C01817=1047.230,-124.087,431.232,169.475,31.897,156.058
C01818=1047.225,-124.336,431.241,169.473,31.897,156.058
C01819=1047.219,-124.586,431.251,169.471,31.897,156.058
C01820=1047.212,-124.836,431.260,169.469,31.897,156.058
C01821=1047.206,-125.086,431.268,169.466,31.896,156.058
C01822=1047.200,-125.335,431.278,169.464,31.897,156.058
C01823=1047.193,-125.585,431.287,169.462,31.897,156.058
C01824=1047.188,-125.835,431.295,169.459,31.897,156.058
C01825=1047.181,-126.085,431.305,169.457,31.897,156.058
C01826=1047.176,-126.335,431.313,169.455,31.897,156.059
C01827=1047.169,-126.584,431.322,169.452,31.897,156.059
C01828=1047.163,-126.834,431.332,169.450,31.896,156.059
C01829=1047.157,-127.084,431.341,169.448,31.897,156.059
C01830=1047.151,-127.333,431.349,169.445,31.896,156.059
C01831=1047.145,-127.583,431.359,169.443,31.897,156.059
C01832=1047.139,-127.833,431.367,169.441,31.897,156.059
C01833=1047.133,-128.082,431.377,169.439,31.896,156.059
C01834=1047.129,-128.332,431.387,169.436,31.895,156.059
C01835=1047.126,-128.582,431.398,169.434,31.894,156.059
C01836=1047.124,-128.832,431.410,169.432,31.892,156.059
C01837=1047.122,-129.082,431.421,169.432,31.890,156.058
C01838=1047.123,-129.332,431.434,169.430,31.887,156.058
C01839=1047.123,-129.583,431.447,169.428,31.883,156.058
C01840=1047.124,-129.832,431.461,169.427,31.880,156.057
C01841=1047.127,-130.083,431.476,169.426,31.876,156.056
C01842=1047.131,-130.334,431.492,169.424,31.871,156.056
C01843=1047.135,-130.585,431.507,169.423,31.866,156.055
C01844=1047.141,-130.835,431.523,169.423,31.861,156.054
C01845=1047.146,-131.085,431.541,169.422,31.854,156.053
C01846=1046.788,-131.108,431.305,169.376,32.030,156.085
C01847=1046.781,-130.858,431.288,169.377,32.036,156.086
C01848=1046.776,-130.609,431.271,169.378,32.042,156.087
C01849=1046.771,-130.358,431.256,169.379,32.047,156.088
C01850=1046.769,-130.107,431.240,169.380,32.051,156.089
C01851=1046.765,-129.857,431.226,169.381,32.055,156.089
C01852=1046.764,-129.607,431.212,169.383,32.059,156.090
C01853=1046.763,-129.356,431.198,169.383,32.063,156.090
C01854=1046.763,-129.106,431.186,169.385,32.065,156.091
C01855=1046.765,-128.856,431.173,169.387,32.068,156.091
C01856=1046.767,-128.606,431.162,169.389,32.070,156.091
C01857=1046.771,-128.356,431.151,169.391,32.071,156.092
C01858=1046.775,-128.106,431.141,169.393,32.072,156.092
C01859=1046.779,-127.856,431.131,169.395,32.072,156.092
C01860=1046.786,-127.607,431.122,169.397,32.073,156.091
C01861=1046.791,-127.357,431.113,169.400,32.072,156.091
C01862=1046.798,-127.107,431.104,169.402,32.072,156.091
C01863=1046.803,-126.858,431.095,169.404,32.072,156.091
C01864=1046.809,-126.608,431.086,169.407,32.072,156.091
C01865=1046.816,-126.358,431.077,169.409,32.072,156.091
C01866=1046.822,-126.108,431.069,169.411,32.072,156.091
C01867=1046.828,-125.859,431.059,169.414,32.072,156.091
C01868=1046.834,-125.609,431.050,169.416,32.072,156.091
C01869=1046.840,-125.359,431.042,169.418,32.072,156.090
C01870=1046.847,-125.109,431.032,169.420,32.072,156.090
C01871=1046.853,-124.860,431.024,169.422,32.072,156.090
C01872=1046.859,-124.610,431.014,169.424,32.072,156.090
C01873=1046.865,-124.360,431.005,169.427,32.072,156.090
C01874=1046.871,-124.110,430.996,169.429,32.072,156.090
C01875=1046.877,-123.861,430.987,169.431,32.072,156.090
C01876=1046.883,-123.611,430.978,169.434,32.073,156.090
C01877=1046.889,-123.361,430.968,169.436,32.072,156.090
C01878=1046.895,-123.111,430.959,169.438,32.072,156.090
C01879=1046.901,-122.862,430.950,169.441,32.073,156.089
C01880=1046.907,-122.612,430.941,169.443,32.072,156.089
C01881=1046.914,-122.362,430.932,169.445,32.073,156.089
C01882=1046.920,-122.112,430.923,169.448,32.073,156.089
C01883=1046.926,-121.862,430.913,169.450,32.073,156.089
C01884=1046.932,-121.613,430.904,169.452,32.073,156.089
C01885=1046.937,-121.363,430.895,169.455,32.073,156.089
C01886=1046.944,-121.113,430.886,169.457,32.073,156.089
C01887=1046.950,-120.864,430.877,169.459,32.073,156.089
C01888=1046.957,-120.614,430.867,169.462,32.073,156.089
C01889=1046.962,-120.365,430.858,169.464,32.074,156.088
C01890=1046.968,-120.114,430.849,169.466,32.074,156.088
C01891=1046.974,-119.864,430.840,169.469,32.074,156.088
C01892=1046.980,-119.615,430.830,169.471,32.074,156.088
C01893=1046.987,-119.365,430.820,169.472,32.074,156.088
C01894=1046.993,-119.115,430.811,169.475,32.075,156.088
C01895=1046.999,-118.866,430.802,169.477,32.075,156.088
C01896=1047.005,-118.616,430.793,169.479,32.074,156.088
C01897=1047.011,-118.366,430.784,169.482,32.075,156.088
C01898=1047.017,-118.116,430.774,169.484,32.075,156.088
C01899=1047.023,-117.866,430.765,169.486,32.075,156.088
C01900=1047.030,-117.617,430.755,169.489,32.076,156.088
C01901=1047.036,-117.367,430.746,169.491,32.075,156.087
C01902=1047.041,-117.118,430.736,169.493,32.075,156.087
C01903=1047.048,-116.868,430.727,169.496,32.076,156.087
C01904=1047.054,-116.618,430.717,169.498,32.076,156.087
C01905=1047.060,-116.368,430.708,169.500,32.076,156.087
C01906=1047.066,-116.119,430.698,169.502,32.076,156.087
C01907=1047.073,-115.833,430.688,169.505,32.077,156.087
C01908=1047.080,-115.547,430.677,169.508,32.077,156.087
C01909=1047.087,-115.262,430.666,169.510,32.077,156.087
C01910=1047.095,-114.976,430.656,169.513,32.077,156.087
C01911=1047.101,-114.726,430.646,169.515,32.077,156.087
C01912=1047.107,-114.476,430.637,169.518,32.078,156.087
C01913=1047.113,-114.226,430.627,169.519,32.078,156.087
C01914=1047.119,-113.977,430.617,169.521,32.078,156.087
C01915=1047.125,-113.727,430.608,169.524,32.079,156.086
C01916=1047.130,-113.477,430.598,169.526,32.079,156.086
C01917=1047.137,-113.228,430.588,169.528,32.079,156.086
C01918=1047.143,-112.978,430.578,169.531,32.079,156.086
C01919=1047.149,-112.729,430.569,169.533,32.080,156.086
C01920=1047.155,-112.479,430.559,169.535,32.080,156.086
C01921=1047.161,-112.229,430.550,169.537,32.080,156.086
C01922=1047.168,-111.979,430.540,169.540,32.080,156.086
C01923=1047.174,-111.729,430.530,169.542,32.081,156.086
C01924=1047.180,-111.480,430.521,169.544,32.081,156.086
C01925=1047.186,-111.230,430.511,169.547,32.081,156.086
C01926=1047.192,-110.980,430.502,169.549,32.082,156.086
C01927=1047.198,-110.730,430.492,169.551,32.082,156.086
C01928=1047.205,-110.481,430.482,169.554,32.082,156.086
C01929=1047.210,-110.231,430.472,169.556,32.082,156.086
C01930=1047.216,-109.981,430.462,169.558,32.083,156.086
C01931=1047.223,-109.731,430.453,169.560,32.083,156.085
C01932=1047.229,-109.481,430.443,169.563,32.083,156.085
C01933=1047.235,-109.232,430.433,169.565,32.083,156.085
C01934=1047.241,-108.983,430.423,169.566,32.084,156.085
C01935=1047.248,-108.733,430.414,169.569,32.084,156.085
C01936=1047.254,-108.483,430.404,169.571,32.085,156.085
C01937=1047.260,-108.233,430.394,169.573,32.085,156.085
C01938=1047.265,-107.983,430.384,169.576,32.086,156.085
C01939=1047.272,-107.734,430.374,169.578,32.086,156.085
C01940=1047.278,-107.484,430.364,169.580,32.086,156.085
C01941=1047.284,-107.234,430.355,169.582,32.086,156.085
C01942=1047.290,-106.984,430.345,169.585,32.087,156.085
C01943=1047.297,-106.735,430.335,169.587,32.087,156.085
C01944=1047.302,-106.485,430.325,169.589,32.088,156.085
C01945=1047.309,-106.235,430.315,169.592,32.088,156.085
C01946=1047.315,-105.986,430.305,169.594,32.088,156.085
C01947=1047.321,-105.736,430.295,169.596,32.089,156.085
C01948=1047.327,-105.486,430.285,169.598,32.089,156.085
C01949=1047.334,-105.236,430.275,169.601,32.090,156.085
C01950=1047.340,-104.987,430.265,169.603,32.090,156.085
C01951=1047.346,-104.737,430.255,169.605,32.090,156.085
C01952=1047.352,-104.487,430.245,169.608,32.091,156.085
C01953=1047.358,-104.238,430.235,169.609,32.092,156.085
C01954=1047.364,-103.988,430.225,169.611,32.092,156.085
C01955=1047.370,-103.738,430.215,169.613,32.092,156.085
C01956=1047.376,-103.488,430.205,169.616,32.092,156.084
C01957=1047.382,-103.239,430.195,169.618,32.093,156.084
C01958=1047.388,-102.989,430.185,169.620,32.093,156.084
C01959=1047.394,-102.739,430.175,169.622,32.094,156.084
C01960=1047.401,-102.489,430.164,169.625,32.095,156.084
C01961=1047.407,-102.240,430.155,169.627,32.095,156.084
C01962=1047.413,-101.990,430.144,169.629,32.095,156.084
C01963=1047.419,-101.740,430.134,169.632,32.096,156.084
C01964=1047.425,-101.491,430.125,169.634,32.096,156.084
C01965=1047.431,-101.241,430.114,169.636,32.097,156.084
C01966=1047.437,-100.991,430.104,169.638,32.097,156.084
C01967=1047.444,-100.742,430.094,169.641,32.098,156.084
C01968=1047.450,-100.491,430.084,169.643,32.098,156.084
C01969=1047.456,-100.242,430.073,169.645,32.098,156.084
C01970=1047.462,-99.992,430.064,169.647,32.099,156.084
C01971=1047.469,-99.705,430.051,169.650,32.100,156.084
C01972=1047.476,-99.419,430.040,169.652,32.101,156.084
C01973=1047.484,-99.132,430.028,169.654,32.101,156.084
C01974=1047.491,-98.846,430.017,169.657,32.101,156.084
C01975=1047.496,-98.597,430.006,169.659,32.102,156.084
C01976=1047.503,-98.346,429.996,169.661,32.102,156.084
C01977=1047.510,-98.097,429.986,169.664,32.103,156.084
C01978=1047.515,-97.847,429.975,169.666,32.103,156.084
C01979=1047.522,-97.598,429.965,169.668,32.104,156.084
C01980=1047.528,-97.347,429.955,169.670,32.105,156.084
C01981=1047.534,-97.098,429.944,169.673,32.105,156.084
C01982=1047.540,-96.848,429.933,169.675,32.106,156.084
C01983=1047.546,-96.598,429.924,169.677,32.106,156.084
C01984=1047.552,-96.349,429.913,169.679,32.107,156.084
C01985=1047.558,-96.099,429.902,169.682,32.108,156.084
C01986=1047.564,-95.849,429.892,169.684,32.108,156.084
C01987=1047.570,-95.599,429.881,169.686,32.109,156.084
C01988=1047.577,-95.350,429.871,169.688,32.109,156.084
C01989=1047.582,-95.100,429.861,169.691,32.110,156.084
C01990=1047.588,-94.851,429.851,169.692,32.110,156.084
C01991=1047.595,-94.601,429.839,169.694,32.111,156.084
C01992=1047.600,-94.351,429.829,169.696,32.112,156.084
C01993=1047.607,-94.101,429.819,169.699,32.113,156.084
C01994=1047.612,-93.852,429.808,169.701,32.113,156.084
C01995=1047.619,-93.602,429.797,169.703,32.114,156.084
C01996=1047.625,-93.352,429.787,169.705,32.115,156.084
C01997=1047.631,-93.102,429.776,169.707,32.115,156.084
C01998=1047.637,-92.853,429.766,169.710,32.116,156.084
C01999=1047.643,-92.603,429.755,169.712,32.117,156.084
C02000=1047.649,-92.353,429.745,169.714,32.117,156.084
C02001=1047.655,-92.104,429.734,169.716,32.118,156.084
C02002=1047.661,-91.854,429.724,169.719,32.119,156.084
C02003=1047.668,-91.604,429.713,169.721,32.119,156.084
C02004=1047.674,-91.355,429.702,169.723,32.120,156.084
C02005=1047.679,-91.105,429.692,169.725,32.121,156.084
C02006=1047.686,-90.855,429.681,169.728,32.121,156.084
C02007=1047.692,-90.605,429.670,169.730,32.122,156.084
C02008=1047.698,-90.356,429.659,169.731,32.123,156.084
C02009=1047.704,-90.107,429.649,169.733,32.123,156.084
C02010=1047.711,-89.857,429.638,169.735,32.124,156.084
C02011=1047.716,-89.607,429.627,169.738,32.125,156.084
C02012=1047.723,-89.357,429.617,169.740,32.125,156.084
C02013=1047.729,-89.107,429.606,169.742,32.126,156.084
C02014=1047.735,-88.858,429.596,169.744,32.127,156.084
C02015=1047.741,-88.608,429.585,169.747,32.127,156.084
C02016=1047.748,-88.358,429.574,169.749,32.128,156.084
C02017=1047.754,-88.109,429.564,169.751,32.129,156.084
C02018=1047.760,-87.859,429.552,169.753,32.129,156.084
C02019=1047.766,-87.609,429.541,169.756,32.130,156.084
C02020=1047.773,-87.360,429.531,169.758,32.131,156.084
C02021=1047.779,-87.110,429.520,169.760,32.132,156.085
C02022=1047.785,-86.860,429.509,169.762,32.132,156.084
C02023=1047.791,-86.611,429.499,169.764,32.133,156.085
C02024=1047.797,-86.361,429.487,169.767,32.134,156.085
C02025=1047.803,-86.111,429.477,169.768,32.135,156.085
C02026=1047.810,-85.861,429.467,169.770,32.135,156.085
C02027=1047.816,-85.612,429.456,169.772,32.136,156.085
C02028=1047.821,-85.362,429.445,169.774,32.137,156.085
C02029=1047.828,-85.112,429.434,169.777,32.137,156.085
C02030=1047.835,-84.863,429.423,169.779,32.138,156.085
C02031=1047.841,-84.613,429.411,169.781,32.139,156.085
C02032=1047.847,-84.364,429.401,169.783,32.140,156.085
C02033=1047.854,-84.114,429.390,169.786,32.141,156.085
C02034=1047.860,-83.864,429.379,169.788,32.141,156.085
C02035=1047.866,-83.580,429.367,169.790,32.142,156.085
C02036=1047.874,-83.295,429.354,169.793,32.143,156.085
C02037=1047.881,-83.011,429.341,169.795,32.144,156.085
C02038=1047.888,-82.726,429.329,169.798,32.145,156.085
C02039=1047.895,-82.476,429.319,169.800,32.146,156.085
C02040=1047.900,-82.227,429.308,169.802,32.146,156.085
C02041=1047.907,-81.977,429.296,169.804,32.147,156.085
C02042=1047.913,-81.728,429.285,169.807,32.148,156.085
C02043=1047.920,-81.478,429.274,169.808,32.148,156.085
C02044=1047.926,-81.229,429.264,169.810,32.149,156.085
C02045=1047.932,-80.978,429.252,169.812,32.150,156.085
C02046=1047.938,-80.729,429.242,169.815,32.151,156.085
C02047=1047.945,-80.479,429.231,169.817,32.151,156.085
C02048=1047.951,-80.230,429.219,169.819,32.152,156.085
C02049=1047.957,-79.980,429.208,169.821,32.153,156.085
C02050=1047.964,-79.731,429.198,169.823,32.154,156.085
C02051=1047.970,-79.481,429.186,169.826,32.155,156.085
C02052=1047.976,-79.231,429.176,169.828,32.156,156.086
C02053=1047.982,-78.981,429.164,169.830,32.157,156.086
C02054=1047.988,-78.732,429.153,169.832,32.158,156.086
C02055=1047.994,-78.482,429.142,169.834,32.158,156.086
C02056=1048.000,-78.232,429.131,169.836,32.159,156.086
C02057=1048.007,-77.983,429.119,169.839,32.160,156.086
C02058=1048.013,-77.733,429.108,169.841,32.161,156.086
C02059=1048.019,-77.483,429.097,169.843,32.162,156.086
C02060=1048.025,-77.234,429.085,169.844,32.163,156.086
C02061=1048.031,-76.984,429.074,169.846,32.164,156.086
C02062=1048.037,-76.734,429.063,169.848,32.165,156.086
C02063=1048.044,-76.485,429.051,169.851,32.166,156.086
C02064=1048.049,-76.235,429.040,169.853,32.166,156.086
C02065=1048.056,-75.985,429.029,169.855,32.167,156.086
C02066=1048.062,-75.736,429.017,169.857,32.168,156.086
C02067=1048.068,-75.486,429.006,169.859,32.169,156.086
C02068=1048.075,-75.236,428.995,169.862,32.170,156.086
C02069=1048.081,-74.987,428.983,169.864,32.171,156.086
C02070=1048.087,-74.737,428.972,169.866,32.172,156.087
C02071=1048.093,-74.487,428.961,169.868,32.173,156.087
C02072=1048.099,-74.238,428.949,169.870,32.173,156.087
C02073=1048.106,-73.988,428.938,169.872,32.174,156.087
C02074=1048.112,-73.739,428.926,169.875,32.175,156.087
C02075=1048.118,-73.489,428.915,169.877,32.177,156.087
C02076=1048.124,-73.240,428.903,169.879,32.178,156.087
C02077=1048.130,-72.989,428.892,169.880,32.178,156.087
C02078=1048.135,-72.740,428.881,169.882,32.179,156.087
C02079=1048.142,-72.490,428.869,169.884,32.181,156.087
C02080=1048.148,-72.241,428.858,169.886,32.182,156.087
C02081=1048.154,-71.991,428.845,169.889,32.183,156.087
C02082=1048.160,-71.741,428.834,169.891,32.184,156.087
C02083=1048.166,-71.492,428.822,169.893,32.185,156.088
C02084=1048.172,-71.242,428.811,169.895,32.186,156.088
C02085=1048.178,-70.993,428.800,169.897,32.187,156.088
C02086=1048.184,-70.743,428.787,169.899,32.188,156.088
C02087=1048.191,-70.493,428.776,169.901,32.189,156.088
C02088=1048.197,-70.244,428.764,169.903,32.190,156.088
C02089=1048.203,-69.994,428.753,169.906,32.191,156.088
C02090=1048.208,-69.744,428.741,169.908,32.192,156.088
C02091=1048.215,-69.494,428.729,169.910,32.193,156.088
C02092=1048.221,-69.245,428.718,169.912,32.194,156.088
C02093=1048.227,-68.995,428.705,169.913,32.195,156.088
C02094=1048.233,-68.745,428.694,169.915,32.196,156.089
C02095=1048.240,-68.496,428.682,169.917,32.197,156.089
C02096=1048.245,-68.246,428.671,169.920,32.198,156.089
C02097=1048.251,-67.996,428.659,169.922,32.200,156.089
C02098=1048.258,-67.747,428.647,169.924,32.201,156.089
C02099=1048.264,-67.465,428.634,169.926,32.201,156.089
C02100=1048.271,-67.183,428.620,169.929,32.203,156.089
C02101=1048.278,-66.900,428.607,169.931,32.204,156.089
C02102=1048.286,-66.618,428.594,169.933,32.205,156.089
C02103=1048.292,-66.368,428.582,169.936,32.206,156.089
C02104=1048.298,-66.118,428.571,169.938,32.208,156.090
C02105=1048.304,-65.869,428.559,169.940,32.209,156.090
C02106=1048.310,-65.619,428.546,169.942,32.210,156.090
C02107=1048.316,-65.369,428.535,169.944,32.211,156.090
C02108=1048.322,-65.120,428.524,169.946,32.212,156.090
C02109=1048.329,-64.871,428.512,169.948,32.213,156.090
C02110=1048.335,-64.621,428.499,169.949,32.214,156.090
C02111=1048.341,-64.371,428.488,169.951,32.215,156.090
C02112=1048.347,-64.122,428.476,169.954,32.216,156.090
C02113=1048.353,-63.872,428.464,169.956,32.218,156.090
C02114=1048.360,-63.622,428.452,169.958,32.218,156.090
C02115=1048.366,-63.372,428.440,169.960,32.219,156.091
C02116=1048.371,-63.123,428.428,169.962,32.221,156.091
C02117=1048.378,-62.873,428.416,169.964,32.222,156.091
C02118=1048.385,-62.624,428.404,169.966,32.223,156.091
C02119=1048.391,-62.374,428.392,169.968,32.224,156.091
C02120=1048.397,-62.124,428.381,169.971,32.225,156.091
C02121=1048.403,-61.875,428.369,169.973,32.226,156.091
C02122=1048.409,-61.625,428.356,169.975,32.227,156.091
C02123=1048.416,-61.376,428.344,169.977,32.229,156.091
C02124=1048.422,-61.126,428.332,169.979,32.230,156.092
C02125=1048.428,-60.876,428.320,169.981,32.231,156.092
C02126=1048.434,-60.627,428.308,169.982,32.232,156.092
C02127=1048.441,-60.377,428.297,169.984,32.233,156.092
C02128=1048.446,-60.127,428.284,169.986,32.234,156.092
C02129=1048.453,-59.878,428.273,169.988,32.235,156.092
C02130=1048.460,-59.628,428.261,169.991,32.236,156.092
C02131=1048.465,-59.379,428.248,169.993,32.238,156.092
C02132=1048.472,-59.129,428.236,169.995,32.238,156.092
C02133=1048.478,-58.880,428.224,169.997,32.240,156.093
C02134=1048.484,-58.630,428.212,169.999,32.241,156.093
C02135=1048.491,-58.380,428.200,170.001,32.242,156.093
C02136=1048.497,-58.130,428.187,170.003,32.243,156.093
C02137=1048.503,-57.881,428.175,170.005,32.244,156.093
C02138=1048.510,-57.631,428.163,170.007,32.246,156.093
C02139=1048.515,-57.382,428.151,170.009,32.246,156.093
C02140=1048.522,-57.132,428.139,170.012,32.248,156.093
C02141=1048.529,-56.883,428.127,170.014,32.249,156.093
C02142=1048.535,-56.633,428.115,170.016,32.250,156.094
C02143=1048.545,-56.216,428.094,170.018,32.252,156.094
C02144=1048.555,-55.799,428.074,170.022,32.254,156.094
C02145=1048.566,-55.381,428.054,170.025,32.256,156.094
C02146=1048.577,-54.964,428.034,170.029,32.258,156.094
C02147=1048.584,-54.714,428.022,170.031,32.259,156.094
C02148=1048.589,-54.465,428.009,170.033,32.260,156.095
C02149=1048.596,-54.215,427.997,170.035,32.261,156.095
C02150=1048.603,-53.965,427.985,170.037,32.262,156.095
C02151=1048.608,-53.716,427.973,170.039,32.264,156.095
C02152=1048.615,-53.467,427.961,170.041,32.265,156.095
C02153=1048.621,-53.217,427.948,170.043,32.266,156.095
C02154=1048.628,-52.968,427.936,170.045,32.267,156.095
C02155=1048.634,-52.718,427.924,170.047,32.268,156.095
C02156=1048.640,-52.468,427.911,170.050,32.269,156.095
C02157=1048.647,-52.219,427.899,170.051,32.271,156.096
C02158=1048.653,-51.969,427.887,170.053,32.272,156.096
C02159=1048.663,-51.606,427.869,170.056,32.274,156.096
C02160=1048.671,-51.243,427.851,170.059,32.275,156.096
C02161=1048.681,-50.880,427.833,170.062,32.277,156.096
C02162=1048.691,-50.517,427.815,170.065,32.279,156.096
C02163=1048.697,-50.267,427.802,170.067,32.280,156.096
C02164=1048.703,-50.017,427.790,170.069,32.282,156.097
C02165=1048.709,-49.767,427.777,170.071,32.283,156.097
C02166=1048.716,-49.518,427.764,170.073,32.284,156.097
C02167=1048.722,-49.268,427.752,170.075,32.285,156.097
C02168=1048.728,-49.018,427.739,170.077,32.287,156.097
C02169=1048.733,-48.768,427.727,170.079,32.288,156.097
C02170=1048.740,-48.520,427.714,170.081,32.289,156.097
C02171=1048.746,-48.270,427.702,170.083,32.291,156.098
C02172=1048.752,-48.020,427.689,170.084,32.292,156.098
C02173=1048.758,-47.771,427.676,170.086,32.294,156.098
C02174=1048.764,-47.522,427.664,170.088,32.294,156.098
C02175=1048.770,-47.272,427.652,170.090,32.296,156.098
C02176=1048.777,-47.022,427.638,170.092,32.297,156.098
C02177=1048.782,-46.773,427.626,170.094,32.299,156.099
C02178=1048.790,-46.522,427.613,170.096,32.300,156.099
C02179=1048.796,-46.273,427.600,170.098,32.301,156.099
C02180=1048.802,-46.023,427.588,170.100,32.303,156.099
C02181=1048.808,-45.774,427.574,170.102,32.304,156.099
C02182=1048.814,-45.524,427.562,170.104,32.306,156.099
C02183=1048.821,-45.274,427.550,170.107,32.307,156.099
C02184=1048.827,-45.025,427.537,170.109,32.308,156.100
C02185=1048.833,-44.775,427.524,170.111,32.310,156.100
C02186=1048.839,-44.526,427.511,170.113,32.311,156.100
C02187=1048.846,-44.276,427.499,170.115,32.312,156.100
C02188=1048.852,-44.027,427.485,170.117,32.313,156.100
C02189=1048.858,-43.777,427.473,170.118,32.315,156.100
C02190=1048.864,-43.527,427.460,170.120,32.316,156.101
C02191=1048.870,-43.278,427.447,170.122,32.318,156.101
C02192=1048.877,-43.029,427.435,170.124,32.319,156.101
C02193=1048.883,-42.779,427.422,170.126,32.320,156.101
C02194=1048.889,-42.529,427.409,170.128,32.322,156.101
C02195=1048.895,-42.279,427.396,170.130,32.323,156.101
C02196=1048.901,-42.030,427.383,170.132,32.324,156.101
C02197=1048.908,-41.781,427.370,170.134,32.326,156.102
C02198=1048.914,-41.531,427.358,170.136,32.327,156.102
C02199=1048.920,-41.281,427.345,170.138,32.328,156.102
C02200=1048.927,-41.032,427.331,170.140,32.330,156.102
C02201=1048.933,-40.782,427.319,170.142,32.331,156.102
C02202=1048.939,-40.532,427.305,170.144,32.333,156.102
C02203=1048.946,-40.283,427.293,170.146,32.334,156.103
C02204=1048.952,-40.034,427.280,170.148,32.335,156.103
C02205=1048.958,-39.784,427.267,170.150,32.336,156.103
C02206=1048.964,-39.534,427.254,170.152,32.338,156.103
C02207=1048.971,-39.285,427.241,170.153,32.339,156.103
C02208=1048.977,-39.035,427.228,170.155,32.341,156.103
C02209=1048.984,-38.786,427.215,170.157,32.342,156.104
C02210=1048.990,-38.536,427.203,170.159,32.344,156.104
C02211=1048.996,-38.286,427.189,170.161,32.345,156.104
C02212=1049.002,-38.037,427.176,170.163,32.347,156.104
C02213=1049.008,-37.787,427.163,170.165,32.348,156.104
C02214=1049.014,-37.537,427.149,170.167,32.350,156.104
C02215=1049.021,-37.288,427.136,170.169,32.351,156.105
C02216=1049.026,-37.038,427.124,170.171,32.353,156.105
C02217=1049.033,-36.789,427.110,170.173,32.354,156.105
C02218=1049.039,-36.539,427.097,170.175,32.356,156.105
C02219=1049.045,-36.290,427.084,170.177,32.357,156.105
C02220=1049.051,-36.040,427.071,170.179,32.359,156.105
C02221=1049.058,-35.790,427.058,170.181,32.360,156.106
C02222=1049.064,-35.541,427.044,170.183,32.361,156.106
C02223=1049.071,-35.261,427.030,170.185,32.363,156.106
C02224=1049.078,-34.980,427.015,170.186,32.364,156.106
C02225=1049.085,-34.699,427.000,170.188,32.366,156.106
C02226=1049.092,-34.419,426.985,170.190,32.368,156.107
C02227=1049.098,-34.170,426.972,170.192,32.369,156.107
C02228=1049.104,-33.920,426.958,170.194,32.371,156.107
C02229=1049.110,-33.671,426.946,170.196,32.372,156.107
C02230=1049.117,-33.421,426.932,170.198,32.374,156.107
C02231=1049.123,-33.171,426.919,170.200,32.375,156.108
C02232=1049.129,-32.922,426.906,170.202,32.377,156.108
C02233=1049.135,-32.673,426.892,170.204,32.378,156.108
C02234=1049.142,-32.423,426.878,170.206,32.380,156.108
C02235=1049.148,-32.173,426.866,170.208,32.381,156.108
C02236=1049.154,-31.923,426.852,170.210,32.383,156.108
C02237=1049.161,-31.673,426.839,170.212,32.384,156.109
C02238=1049.167,-31.424,426.825,170.214,32.386,156.109
C02239=1049.173,-31.175,426.812,170.216,32.387,156.109
C02240=1049.179,-30.926,426.799,170.218,32.388,156.109
C02241=1049.186,-30.676,426.785,170.219,32.390,156.109
C02242=1049.192,-30.426,426.772,170.221,32.391,156.109
C02243=1049.198,-30.177,426.758,170.223,32.393,156.110
C02244=1049.204,-29.926,426.745,170.225,32.394,156.110
C02245=1049.211,-29.677,426.732,170.227,32.396,156.110
C02246=1049.217,-29.428,426.719,170.229,32.398,156.110
C02247=1049.223,-29.178,426.705,170.231,32.399,156.110
C02248=1049.230,-28.928,426.692,170.233,32.401,156.111
C02249=1049.236,-28.679,426.678,170.235,32.402,156.111
C02250=1049.242,-28.430,426.665,170.236,32.404,156.111
C02251=1049.248,-28.180,426.651,170.238,32.405,156.111
C02252=1049.255,-27.930,426.638,170.240,32.407,156.111
C02253=1049.261,-27.680,426.624,170.242,32.408,156.112
C02254=1049.268,-27.431,426.611,170.244,32.409,156.112
C02255=1049.274,-27.182,426.598,170.246,32.411,156.112
C02256=1049.281,-26.932,426.584,170.248,32.412,156.112
C02257=1049.286,-26.682,426.570,170.250,32.414,156.112
C02258=1049.292,-26.433,426.557,170.252,32.416,156.113
C02259=1049.299,-26.183,426.543,170.253,32.417,156.113
C02260=1049.305,-25.934,426.529,170.255,32.419,156.113
C02261=1049.311,-25.684,426.516,170.257,32.420,156.113
C02262=1049.318,-25.435,426.502,170.259,32.422,156.113
C02263=1049.323,-25.185,426.488,170.261,32.424,156.114
C02264=1049.330,-24.936,426.475,170.263,32.425,156.114
C02265=1049.336,-24.686,426.460,170.264,32.427,156.114
C02266=1049.342,-24.437,426.447,170.266,32.428,156.114
C02267=1049.348,-24.187,426.434,170.268,32.430,156.114
C02268=1049.354,-23.937,426.420,170.270,32.432,156.115
C02269=1049.360,-23.688,426.406,170.272,32.433,156.115
C02270=1049.367,-23.439,426.392,170.274,32.435,156.115
C02271=1049.373,-23.189,426.378,170.276,32.437,156.115
C02272=1049.379,-22.940,426.365,170.278,32.438,156.115
C02273=1049.385,-22.689,426.351,170.280,32.440,156.116
C02274=1049.391,-22.440,426.337,170.282,32.441,156.116
C02275=1049.398,-22.191,426.323,170.284,32.443,156.116
C02276=1049.404,-21.941,426.309,170.285,32.444,156.116
C02277=1049.410,-21.692,426.296,170.287,32.446,156.116
C02278=1049.416,-21.442,426.282,170.288,32.447,156.117
C02279=1049.423,-21.192,426.268,170.290,32.449,156.117
C02280=1049.430,-20.943,426.254,170.292,32.451,156.117
C02281=1049.435,-20.693,426.240,170.294,32.452,156.117
C02282=1049.441,-20.444,426.227,170.296,32.454,156.117
C02283=1049.447,-20.194,426.213,170.298,32.456,156.118
C02284=1049.454,-19.945,426.199,170.300,32.457,156.118
C02285=1049.461,-19.695,426.185,170.302,32.459,156.118
C02286=1049.466,-19.446,426.171,170.303,32.460,156.118
C02287=1049.473,-19.165,426.155,170.306,32.462,156.119
C02288=1049.480,-18.883,426.140,170.308,32.464,156.119
C02289=1049.488,-18.602,426.124,170.310,32.466,156.119
C02290=1049.495,-18.321,426.108,170.312,32.468,156.119
C02291=1049.501,-18.071,426.094,170.314,32.469,156.120
C02292=1049.508,-17.822,426.080,170.316,32.471,156.120
C02293=1049.513,-17.572,426.066,170.318,32.472,156.120
C02294=1049.520,-17.322,426.053,170.320,32.474,156.120
C02295=1049.527,-17.074,426.039,170.321,32.476,156.120
C02296=1049.533,-16.823,426.024,170.323,32.477,156.121
C02297=1049.539,-16.574,426.011,170.324,32.479,156.121
C02298=1049.545,-16.325,425.996,170.326,32.481,156.121
C02299=1049.552,-16.075,425.983,170.328,32.482,156.121
C02300=1049.558,-15.826,425.968,170.330,32.484,156.121
C02301=1049.564,-15.576,425.955,170.332,32.486,156.122
C02302=1049.570,-15.326,425.940,170.334,32.487,156.122
C02303=1049.577,-15.077,425.926,170.336,32.489,156.122
C02304=1049.583,-14.827,425.912,170.337,32.491,156.122
C02305=1049.590,-14.578,425.898,170.339,32.492,156.123
C02306=1049.595,-14.328,425.884,170.341,32.494,156.123
C02307=1049.602,-14.079,425.869,170.343,32.496,156.123
C02308=1049.608,-13.829,425.856,170.345,32.497,156.123
C02309=1049.614,-13.580,425.841,170.347,32.499,156.123
C02310=1049.620,-13.330,425.827,170.349,32.501,156.124
C02311=1049.627,-13.081,425.813,170.350,32.503,156.124
C02312=1049.633,-12.831,425.799,170.352,32.504,156.124
C02313=1049.639,-12.582,425.784,170.354,32.506,156.124
C02314=1049.645,-12.332,425.771,170.356,32.508,156.125
C02315=1049.652,-12.083,425.756,170.358,32.509,156.125
C02316=1049.657,-11.833,425.742,170.359,32.511,156.125
C02317=1049.663,-11.583,425.727,170.361,32.513,156.125
C02318=1049.670,-11.334,425.714,170.362,32.515,156.126
C02319=1049.676,-11.084,425.699,170.364,32.516,156.126
C02320=1049.682,-10.835,425.684,170.366,32.518,156.126
C02321=1049.689,-10.586,425.670,170.368,32.520,156.126
C02322=1049.695,-10.336,425.655,170.370,32.521,156.126
C02323=1049.700,-10.086,425.642,170.372,32.523,156.127
C02324=1049.708,-9.837,425.627,170.374,32.524,156.127
C02325=1049.714,-9.587,425.612,170.375,32.526,156.127
C02326=1049.719,-9.338,425.598,170.377,32.528,156.127
C02327=1049.727,-9.088,425.584,170.379,32.530,156.128
C02328=1049.732,-8.839,425.570,170.381,32.531,156.128
C02329=1049.738,-8.589,425.555,170.383,32.533,156.128
C02330=1049.745,-8.339,425.540,170.385,32.535,156.128
C02331=1049.751,-8.091,425.526,170.386,32.536,156.129
C02332=1049.757,-7.841,425.512,170.388,32.538,156.129
C02333=1049.763,-7.592,425.498,170.390,32.540,156.129
C02334=1049.770,-7.342,425.483,170.392,32.542,156.129
C02335=1049.776,-7.092,425.469,170.394,32.543,156.130
C02336=1049.782,-6.843,425.454,170.396,32.545,156.130
C02337=1049.789,-6.593,425.439,170.396,32.547,156.130
C02338=1049.796,-6.344,425.425,170.398,32.549,156.130
C02339=1049.801,-6.094,425.411,170.400,32.550,156.131
C02340=1049.808,-5.845,425.396,170.402,32.552,156.131
C02341=1049.814,-5.595,425.381,170.404,32.554,156.131
C02342=1049.820,-5.346,425.368,170.406,32.555,156.131
C02343=1049.826,-5.096,425.353,170.407,32.557,156.131
C02344=1049.833,-4.847,425.338,170.409,32.559,156.132
C02345=1049.839,-4.598,425.324,170.411,32.561,156.132
C02346=1049.846,-4.348,425.309,170.413,32.562,156.132
C02347=1049.852,-4.098,425.295,170.415,32.564,156.132
C02348=1049.858,-3.848,425.280,170.417,32.566,156.133
C02349=1049.865,-3.600,425.266,170.418,32.568,156.133
C02350=1049.871,-3.350,425.251,170.420,32.569,156.133
C02351=1049.878,-3.067,425.235,170.422,32.571,156.133
C02352=1049.884,-2.784,425.217,170.424,32.573,156.134
C02353=1049.892,-2.501,425.200,170.426,32.575,156.134
C02354=1049.898,-2.218,425.184,170.428,32.577,156.134
C02355=1049.905,-1.969,425.169,170.430,32.579,156.135
C02356=1049.911,-1.719,425.155,170.432,32.581,156.135
C02357=1049.917,-1.470,425.140,170.434,32.583,156.135
C02358=1049.923,-1.221,425.125,170.435,32.585,156.135
C02359=1049.929,-0.971,425.110,170.436,32.586,156.136
C02360=1049.935,-0.722,425.095,170.438,32.588,156.136
C02361=1049.942,-0.472,425.081,170.440,32.590,156.136
C02362=1049.948,-0.223,425.066,170.442,32.592,156.136
C02363=1049.954,0.027,425.051,170.444,32.594,156.137
C02364=1049.960,0.276,425.036,170.445,32.595,156.137
C02365=1049.967,0.526,425.021,170.447,32.597,156.137
C02366=1049.973,0.775,425.006,170.449,32.599,156.137
C02367=1049.979,1.024,424.992,170.451,32.601,156.138
C02368=1049.985,1.274,424.977,170.453,32.603,156.138
C02369=1049.991,1.524,424.961,170.454,32.605,156.138
C02370=1049.997,1.774,424.946,170.456,32.606,156.138
C02371=1050.003,2.022,424.932,170.458,32.608,156.139
C02372=1050.009,2.272,424.917,170.460,32.610,156.139
C02373=1050.016,2.522,424.902,170.461,32.612,156.139
C02374=1050.022,2.771,424.887,170.463,32.614,156.139
C02375=1050.028,3.020,424.872,170.465,32.616,156.140
C02376=1050.034,3.270,424.857,170.467,32.617,156.140
C02377=1050.041,3.520,424.842,170.469,32.619,156.140
C02378=1050.047,3.769,424.827,170.470,32.621,156.141
C02379=1050.053,4.018,424.813,170.472,32.623,156.141
C02380=1050.059,4.268,424.798,170.474,32.625,156.141
C02381=1050.066,4.518,424.783,170.475,32.626,156.141
C02382=1050.071,4.768,424.767,170.477,32.628,156.142
C02383=1050.078,5.017,424.752,170.478,32.630,156.142
C02384=1050.084,5.266,424.737,170.480,32.632,156.142
C02385=1050.090,5.515,424.722,170.482,32.634,156.142
C02386=1050.096,5.765,424.707,170.484,32.636,156.143
C02387=1050.103,6.015,424.692,170.485,32.637,156.143
C02388=1050.109,6.264,424.677,170.487,32.639,156.143
C02389=1050.115,6.513,424.663,170.489,32.641,156.143
C02390=1050.122,6.762,424.647,170.491,32.643,156.144
C02391=1050.128,7.012,424.632,170.493,32.645,156.144
C02392=1050.134,7.262,424.617,170.494,32.647,156.144
C02393=1050.140,7.512,424.602,170.496,32.648,156.144
C02394=1050.146,7.761,424.587,170.498,32.650,156.145
C02395=1050.153,8.010,424.571,170.500,32.652,156.145
C02396=1050.159,8.259,424.556,170.501,32.654,156.145
C02397=1050.165,8.509,424.541,170.503,32.656,156.146
C02398=1050.172,8.758,424.527,170.505,32.658,156.146
C02399=1050.178,9.008,424.512,170.507,32.659,156.146
C02400=1050.185,9.257,424.496,170.508,32.661,156.146
C02401=1050.190,9.507,424.480,170.510,32.663,156.147
C02402=1050.197,9.757,424.465,170.512,32.665,156.147
C02403=1050.203,10.006,424.450,170.514,32.667,156.147
C02404=1050.210,10.255,424.435,170.516,32.669,156.147
C02405=1050.216,10.504,424.420,170.517,32.670,156.148
C02406=1050.222,10.754,424.405,170.518,32.672,156.148
C02407=1050.229,11.003,424.390,170.520,32.674,156.148
C02408=1050.234,11.253,424.374,170.522,32.676,156.148
C02409=1050.241,11.503,424.359,170.523,32.678,156.149
C02410=1050.247,11.752,424.343,170.525,32.679,156.149
C02411=1050.254,12.001,424.329,170.527,32.681,156.149
C02412=1050.260,12.251,424.314,170.529,32.683,156.149
C02413=1050.267,12.500,424.298,170.530,32.685,156.150
C02414=1050.273,12.750,424.283,170.532,32.687,156.150
C02415=1050.280,13.034,424.266,170.534,32.689,156.150
C02416=1050.288,13.320,424.248,170.536,32.691,156.151
C02417=1050.295,13.604,424.231,170.538,32.693,156.151
C02418=1050.302,13.889,424.213,170.540,32.695,156.151
C02419=1050.309,14.138,424.197,170.542,32.697,156.151
C02420=1050.315,14.388,424.182,170.544,32.699,156.152
C02421=1050.320,14.637,424.167,170.545,32.700,156.152
C02422=1050.327,14.886,424.152,170.547,32.702,156.152
C02423=1050.333,15.136,424.136,170.549,32.704,156.153
C02424=1050.339,15.385,424.120,170.551,32.706,156.153
C02425=1050.345,15.635,424.105,170.552,32.708,156.153
C02426=1050.352,15.884,424.089,170.554,32.710,156.153
C02427=1050.358,16.134,424.074,170.556,32.712,156.154
C02428=1050.364,16.383,424.058,170.558,32.714,156.154
C02429=1050.370,16.633,424.043,170.559,32.716,156.154
C02430=1050.376,16.882,424.027,170.561,32.718,156.155
C02431=1050.383,17.132,424.012,170.563,32.719,156.155
C02432=1050.389,17.381,423.996,170.563,32.721,156.155
C02433=1050.395,17.631,423.981,170.565,32.723,156.155
C02434=1050.402,17.880,423.965,170.567,32.725,156.156
C02435=1050.407,18.130,423.949,170.569,32.727,156.156
C02436=1050.414,18.379,423.934,170.570,32.729,156.156
C02437=1050.421,18.628,423.918,170.572,32.731,156.156
C02438=1050.426,18.878,423.903,170.574,32.733,156.157
C02439=1050.433,19.127,423.887,170.576,32.735,156.157
C02440=1050.439,19.377,423.871,170.577,32.736,156.157
C02441=1050.445,19.626,423.856,170.579,32.738,156.158
C02442=1050.451,19.876,423.840,170.581,32.740,156.158
C02443=1050.458,20.125,423.824,170.582,32.742,156.158
C02444=1050.464,20.374,423.808,170.584,32.744,156.159
C02445=1050.470,20.624,423.793,170.586,32.746,156.159
C02446=1050.476,20.873,423.777,170.588,32.748,156.159
C02447=1050.483,21.122,423.761,170.589,32.750,156.159
C02448=1050.488,21.372,423.746,170.591,32.752,156.160
C02449=1050.495,21.621,423.730,170.593,32.754,156.160
C02450=1050.501,21.871,423.714,170.594,32.756,156.160
C02451=1050.507,22.120,423.699,170.596,32.758,156.161
C02452=1050.513,22.370,423.683,170.598,32.760,156.161
C02453=1050.520,22.619,423.667,170.600,32.761,156.161
C02454=1050.526,22.869,423.651,170.601,32.763,156.161
C02455=1050.532,23.118,423.635,170.603,32.765,156.162
C02456=1050.538,23.367,423.620,170.605,32.767,156.162
C02457=1050.545,23.617,423.603,170.606,32.769,156.162
C02458=1050.551,23.867,423.588,170.608,32.771,156.163
C02459=1050.557,24.116,423.572,170.610,32.773,156.163
C02460=1050.564,24.365,423.556,170.612,32.775,156.163
C02461=1050.570,24.615,423.540,170.613,32.777,156.163
C02462=1050.576,24.865,423.524,170.614,32.779,156.164
C02463=1050.582,25.114,423.509,170.616,32.781,156.164
C02464=1050.588,25.363,423.492,170.617,32.783,156.164
C02465=1050.595,25.612,423.477,170.619,32.785,156.165
C02466=1050.601,25.861,423.460,170.621,32.787,156.165
C02467=1050.607,26.111,423.445,170.623,32.788,156.165
C02468=1050.614,26.361,423.429,170.624,32.790,156.165
C02469=1050.620,26.610,423.413,170.626,32.792,156.166
C02470=1050.626,26.859,423.397,170.628,32.794,156.166
C02471=1050.632,27.109,423.381,170.629,32.796,156.166
C02472=1050.638,27.358,423.364,170.631,32.798,156.167
C02473=1050.645,27.608,423.349,170.633,32.800,156.167
C02474=1050.651,27.857,423.333,170.634,32.802,156.167
C02475=1050.657,28.106,423.318,170.636,32.804,156.167
C02476=1050.664,28.356,423.301,170.638,32.806,156.168
C02477=1050.670,28.606,423.285,170.640,32.808,156.168
C02478=1050.676,28.855,423.268,170.641,32.810,156.168
C02479=1050.683,29.140,423.250,170.643,32.812,156.169
C02480=1050.690,29.427,423.232,170.645,32.815,156.169
C02481=1050.697,29.713,423.213,170.647,32.817,156.169
C02482=1050.704,29.998,423.195,170.649,32.819,156.170
C02483=1050.710,30.248,423.178,170.651,32.821,156.170
C02484=1050.717,30.498,423.162,170.652,32.823,156.170
C02485=1050.723,30.747,423.146,170.654,32.825,156.171
C02486=1050.729,30.996,423.130,170.656,32.827,156.171
C02487=1050.735,31.246,423.114,170.657,32.829,156.171
C02488=1050.741,31.495,423.097,170.659,32.831,156.172
C02489=1050.747,31.744,423.081,170.661,32.833,156.172
C02490=1050.754,31.993,423.065,170.662,32.835,156.172
C02491=1050.760,32.243,423.049,170.664,32.837,156.172
C02492=1050.766,32.493,423.032,170.666,32.839,156.173
C02493=1050.772,32.742,423.016,170.667,32.841,156.173
C02494=1050.778,32.991,423.000,170.669,32.843,156.173
C02495=1050.785,33.240,422.984,170.671,32.845,156.174
C02496=1050.791,33.491,422.968,170.672,32.847,156.174
C02497=1050.797,33.740,422.951,170.673,32.849,156.174
C02498=1050.803,33.989,422.935,170.675,32.851,156.175
C02499=1050.809,34.239,422.919,170.677,32.853,156.175
C02500=1050.815,34.488,422.903,170.678,32.855,156.175
C02501=1050.823,34.738,422.887,170.680,32.857,156.176
C02502=1050.829,34.987,422.870,170.682,32.859,156.176
C02503=1050.834,35.236,422.854,170.683,32.861,156.176
C02504=1050.841,35.485,422.837,170.685,32.862,156.176
C02505=1050.847,35.735,422.821,170.687,32.864,156.177
C02506=1050.853,35.984,422.804,170.688,32.866,156.177
C02507=1050.860,36.234,422.789,170.690,32.868,156.177
C02508=1050.866,36.483,422.772,170.692,32.870,156.178
C02509=1050.872,36.733,422.756,170.693,32.872,156.178
C02510=1050.878,36.982,422.739,170.695,32.874,156.178
C02511=1050.885,37.231,422.723,170.697,32.876,156.178
C02512=1050.891,37.480,422.706,170.698,32.878,156.179
C02513=1050.897,37.730,422.690,170.700,32.880,156.179
C02514=1050.903,37.980,422.673,170.702,32.882,156.179
C02515=1050.909,38.229,422.657,170.703,32.884,156.180
C02516=1050.915,38.478,422.640,170.705,32.886,156.180
C02517=1050.922,38.728,422.624,170.707,32.888,156.180
C02518=1050.928,38.977,422.607,170.708,32.890,156.181
C02519=1050.934,39.227,422.591,170.710,32.892,156.181
C02520=1050.940,39.475,422.574,170.712,32.894,156.181
C02521=1050.947,39.725,422.557,170.713,32.896,156.182
C02522=1050.953,39.975,422.541,170.715,32.898,156.182
C02523=1050.959,40.223,422.524,170.717,32.900,156.182
C02524=1050.965,40.473,422.508,170.718,32.902,156.183
C02525=1050.971,40.723,422.491,170.720,32.904,156.183
C02526=1050.978,40.972,422.474,170.722,32.906,156.183
C02527=1050.983,41.221,422.458,170.723,32.909,156.184
C02528=1050.990,41.471,422.441,170.725,32.911,156.184
C02529=1050.996,41.720,422.424,170.727,32.913,156.184
C02530=1051.002,41.969,422.408,170.728,32.915,156.184
C02531=1051.008,42.218,422.392,170.730,32.917,156.185
C02532=1051.014,42.468,422.374,170.732,32.919,156.185
C02533=1051.020,42.717,422.358,170.733,32.921,156.185
C02534=1051.026,42.967,422.342,170.735,32.923,156.186
C02535=1051.033,43.216,422.324,170.737,32.925,156.186
C02536=1051.039,43.466,422.308,170.738,32.927,156.186
C02537=1051.045,43.714,422.291,170.740,32.929,156.187
C02538=1051.052,43.964,422.274,170.742,32.931,156.187
C02539=1051.057,44.214,422.257,170.743,32.933,156.187
C02540=1051.063,44.463,422.241,170.744,32.935,156.188
C02541=1051.069,44.712,422.224,170.745,32.937,156.188
C02542=1051.075,44.962,422.206,170.747,32.940,156.188
C02543=1051.083,45.248,422.188,170.749,32.942,156.189
C02544=1051.089,45.533,422.168,170.751,32.944,156.189
C02545=1051.096,45.820,422.149,170.753,32.947,156.189
C02546=1051.103,46.105,422.130,170.755,32.949,156.190
C02547=1051.109,46.355,422.113,170.756,32.951,156.190
C02548=1051.116,46.605,422.095,170.758,32.953,156.190
C02549=1051.122,46.853,422.078,170.760,32.955,156.191
C02550=1051.127,47.103,422.061,170.761,32.957,156.191
C02551=1051.134,47.352,422.044,170.763,32.959,156.191
C02552=1051.140,47.602,422.028,170.764,32.961,156.192
C02553=1051.145,47.851,422.010,170.766,32.963,156.192
C02554=1051.152,48.101,421.994,170.768,32.965,156.192
C02555=1051.158,48.350,421.977,170.769,32.967,156.193
C02556=1051.164,48.600,421.960,170.771,32.970,156.193
C02557=1051.170,48.849,421.943,170.773,32.972,156.193
C02558=1051.177,49.097,421.926,170.774,32.974,156.194
C02559=1051.182,49.348,421.908,170.776,32.976,156.194
C02560=1051.189,49.596,421.891,170.778,32.978,156.194
C02561=1051.195,49.846,421.875,170.779,32.980,156.195
C02562=1051.201,50.096,421.857,170.781,32.982,156.195
C02563=1051.207,50.344,421.840,170.782,32.984,156.195
C02564=1051.213,50.594,421.824,170.784,32.987,156.196
C02565=1051.219,50.843,421.806,170.786,32.989,156.196
C02566=1051.225,51.092,421.789,170.787,32.990,156.196
C02567=1051.232,51.342,421.772,170.789,32.993,156.197
C02568=1051.237,51.591,421.755,170.791,32.995,156.197
C02569=1051.244,51.841,421.738,170.792,32.996,156.197
C02570=1051.250,52.090,421.721,170.794,32.998,156.198
C02571=1051.256,52.340,421.703,170.796,33.001,156.198
C02572=1051.262,52.588,421.686,170.797,33.003,156.198
C02573=1051.268,52.838,421.670,170.799,33.005,156.199
C02574=1051.275,53.088,421.652,170.800,33.007,156.199
C02575=1051.281,53.336,421.635,170.802,33.009,156.199
C02576=1051.287,53.586,421.617,170.804,33.011,156.200
C02577=1051.293,53.835,421.601,170.805,33.013,156.200
C02578=1051.300,54.085,421.584,170.807,33.015,156.200
C02579=1051.305,54.334,421.566,170.809,33.017,156.201
C02580=1051.312,54.583,421.549,170.810,33.019,156.201
C02581=1051.318,54.833,421.533,170.812,33.022,156.201
C02582=1051.324,55.082,421.515,170.814,33.024,156.202
C02583=1051.330,55.331,421.498,170.815,33.026,156.202
C02584=1051.337,55.581,421.480,170.817,33.028,156.202
C02585=1051.343,55.830,421.463,170.819,33.030,156.203
C02586=1051.349,56.080,421.446,170.820,33.032,156.203
C02587=1051.355,56.329,421.429,170.822,33.034,156.203
C02588=1051.362,56.578,421.411,170.823,33.035,156.203
C02589=1051.367,56.827,421.394,170.825,33.037,156.204
C02590=1051.374,57.077,421.376,170.827,33.040,156.204
C02591=1051.380,57.326,421.360,170.828,33.042,156.205
C02592=1051.386,57.576,421.342,170.830,33.044,156.205
C02593=1051.392,57.824,421.325,170.832,33.046,156.205
C02594=1051.399,58.074,421.307,170.833,33.048,156.205
C02595=1051.405,58.323,421.290,170.835,33.050,156.206
C02596=1051.412,58.572,421.273,170.837,33.052,156.206
C02597=1051.418,58.822,421.255,170.838,33.054,156.206
C02598=1051.424,59.071,421.238,170.840,33.056,156.207
C02599=1051.430,59.320,421.220,170.842,33.058,156.207
C02600=1051.436,59.570,421.204,170.843,33.060,156.207
C02601=1051.443,59.819,421.186,170.845,33.062,156.208
C02602=1051.449,60.068,421.169,170.846,33.064,156.208
C02603=1051.455,60.318,421.152,170.848,33.066,156.208
C02604=1051.461,60.567,421.134,170.850,33.069,156.209
C02605=1051.468,60.816,421.117,170.851,33.070,156.209
C02606=1051.474,61.066,421.099,170.853,33.073,156.209
C02607=1051.482,61.352,421.079,170.855,33.075,156.210
C02608=1051.489,61.637,421.059,170.857,33.077,156.210
C02609=1051.496,61.923,421.039,170.859,33.079,156.210
C02610=1051.503,62.209,421.019,170.861,33.082,156.211
C02611=1051.509,62.457,421.002,170.862,33.084,156.211
C02612=1051.515,62.707,420.984,170.863,33.086,156.211
C02613=1051.522,62.957,420.967,170.865,33.088,156.212
C02614=1051.528,63.205,420.950,170.866,33.090,156.212
C02615=1051.534,63.455,420.932,170.868,33.092,156.212
C02616=1051.541,63.705,420.914,170.869,33.094,156.213
C02617=1051.547,63.954,420.897,170.871,33.096,156.213
C02618=1051.554,64.203,420.879,170.873,33.098,156.213
C02619=1051.560,64.453,420.861,170.874,33.100,156.214
C02620=1051.565,64.702,420.844,170.876,33.102,156.214
C02621=1051.572,64.951,420.826,170.878,33.104,156.214
C02622=1051.578,65.200,420.808,170.879,33.106,156.215
C02623=1051.584,65.449,420.790,170.881,33.108,156.215
C02624=1051.591,65.699,420.773,170.883,33.110,156.215
C02625=1051.596,65.948,420.755,170.884,33.113,156.216
C02626=1051.603,66.198,420.737,170.886,33.115,156.216
C02627=1051.609,66.447,420.720,170.887,33.117,156.216
C02628=1051.615,66.695,420.702,170.889,33.119,156.217
C02629=1051.621,66.945,420.684,170.891,33.121,156.217
C02630=1051.627,67.194,420.666,170.892,33.123,156.217
C02631=1051.634,67.444,420.649,170.894,33.125,156.218
C02632=1051.640,67.693,420.631,170.896,33.127,156.218
C02633=1051.645,67.942,420.614,170.897,33.129,156.218
C02634=1051.652,68.192,420.595,170.899,33.131,156.219
C02635=1051.659,68.441,420.578,170.900,33.133,156.219
C02636=1051.664,68.690,420.560,170.902,33.136,156.219
C02637=1051.670,68.940,420.542,170.904,33.138,156.220
C02638=1051.677,69.189,420.523,170.905,33.140,156.220
C02639=1051.683,69.438,420.506,170.907,33.142,156.220
C02640=1051.689,69.687,420.488,170.909,33.144,156.221
C02641=1051.695,69.937,420.471,170.910,33.146,156.221
C02642=1051.701,70.185,420.452,170.912,33.148,156.221
C02643=1051.707,70.435,420.434,170.914,33.150,156.222
C02644=1051.713,70.685,420.416,170.915,33.152,156.222
C02645=1051.719,70.933,420.398,170.917,33.155,156.223
C02646=1051.726,71.183,420.381,170.918,33.157,156.223
C02647=1051.732,71.433,420.363,170.920,33.159,156.223
C02648=1051.738,71.681,420.345,170.922,33.161,156.223
C02649=1051.744,71.931,420.327,170.923,33.163,156.224
C02650=1051.750,72.180,420.309,170.925,33.165,156.224
C02651=1051.757,72.430,420.290,170.927,33.167,156.225
C02652=1051.762,72.679,420.272,170.928,33.169,156.225
C02653=1051.768,72.928,420.255,170.930,33.171,156.225
C02654=1051.775,73.178,420.236,170.931,33.174,156.226
C02655=1051.781,73.426,420.219,170.933,33.176,156.226
C02656=1051.787,73.675,420.200,170.935,33.178,156.226
C02657=1051.793,73.925,420.182,170.936,33.180,156.227
C02658=1051.800,74.175,420.164,170.938,33.182,156.227
C02659=1051.805,74.423,420.146,170.940,33.184,156.227
C02660=1051.812,74.673,420.128,170.941,33.186,156.228
C02661=1051.818,74.922,420.110,170.943,33.188,156.228
C02662=1051.823,75.171,420.092,170.944,33.191,156.228
C02663=1051.830,75.420,420.073,170.946,33.193,156.229
C02664=1051.836,75.670,420.055,170.948,33.195,156.229
C02665=1051.842,75.919,420.037,170.949,33.197,156.229
C02666=1051.849,76.169,420.019,170.951,33.199,156.230
C02667=1051.854,76.417,420.001,170.953,33.201,156.230
C02668=1051.861,76.667,419.983,170.954,33.203,156.230
C02669=1051.867,76.916,419.964,170.956,33.205,156.231
C02670=1051.873,77.166,419.946,170.957,33.207,156.231
C02671=1051.880,77.451,419.925,170.959,33.210,156.231
C02672=1051.888,77.737,419.905,170.961,33.212,156.232
C02673=1051.894,78.022,419.883,170.963,33.214,156.232
C02674=1051.901,78.307,419.863,170.965,33.217,156.233
C02675=1051.908,78.557,419.845,170.967,33.219,156.233
C02676=1051.914,78.806,419.826,170.968,33.222,156.233
C02677=1051.919,79.055,419.809,170.970,33.224,156.234
C02678=1051.925,79.305,419.789,170.971,33.225,156.234
C02679=1051.932,79.554,419.771,170.973,33.228,156.234
C02680=1051.938,79.804,419.753,170.975,33.230,156.235
C02681=1051.944,80.053,419.734,170.976,33.232,156.235
C02682=1051.950,80.301,419.716,170.978,33.235,156.235
C02683=1051.955,80.551,419.697,170.980,33.237,156.236
C02684=1051.962,80.800,419.679,170.981,33.239,156.236
C02685=1051.968,81.049,419.660,170.983,33.241,156.237
C02686=1051.974,81.299,419.642,170.984,33.243,156.237
C02687=1051.980,81.548,419.624,170.986,33.245,156.237
C02688=1051.986,81.797,419.605,170.988,33.248,156.238
C02689=1051.992,82.047,419.587,170.989,33.250,156.238
C02690=1051.998,82.296,419.568,170.991,33.252,156.238
C02691=1052.005,82.545,419.549,170.993,33.254,156.239
C02692=1052.010,82.794,419.532,170.994,33.256,156.239
C02693=1052.016,83.044,419.513,170.996,33.258,156.239
C02694=1052.022,83.293,419.494,170.997,33.260,156.240
C02695=1052.029,83.542,419.475,170.999,33.263,156.240
C02696=1052.035,83.792,419.457,171.001,33.265,156.240
C02697=1052.041,84.041,419.439,171.002,33.267,156.241
C02698=1052.046,84.289,419.420,171.004,33.269,156.241
C02699=1052.053,84.538,419.401,171.006,33.271,156.241
C02700=1052.059,84.788,419.383,171.007,33.273,156.242
C02701=1052.065,85.037,419.365,171.009,33.275,156.242
C02702=1052.072,85.286,419.346,171.010,33.278,156.243
C02703=1052.078,85.536,419.327,171.012,33.280,156.243
C02704=1052.084,85.785,419.308,171.014,33.282,156.243
C02705=1052.090,86.035,419.290,171.016,33.284,156.244
C02706=1052.096,86.283,419.272,171.018,33.286,156.244
C02707=1052.102,86.533,419.253,171.020,33.288,156.244
C02708=1052.108,86.782,419.234,171.021,33.290,156.245
C02709=1052.114,87.031,419.215,171.023,33.293,156.245
C02710=1052.121,87.280,419.197,171.025,33.295,156.245
C02711=1052.126,87.530,419.178,171.026,33.297,156.246
C02712=1052.133,87.779,419.159,171.028,33.299,156.246
C02713=1052.139,88.028,419.141,171.029,33.301,156.246
C02714=1052.146,88.277,419.122,171.031,33.303,156.247
C02715=1052.151,88.527,419.103,171.033,33.305,156.247
C02716=1052.158,88.776,419.084,171.034,33.307,156.247
C02717=1052.164,89.025,419.066,171.036,33.310,156.248
C02718=1052.171,89.274,419.047,171.038,33.312,156.248
C02719=1052.176,89.524,419.028,171.039,33.314,156.248
C02720=1052.182,89.772,419.009,171.041,33.316,156.249
C02721=1052.188,90.022,418.991,171.043,33.318,156.249
C02722=1052.195,90.271,418.973,171.044,33.320,156.249
C02723=1052.200,90.520,418.954,171.046,33.322,156.250
C02724=1052.207,90.769,418.935,171.048,33.325,156.250
C02725=1052.212,91.019,418.916,171.049,33.327,156.251
C02726=1052.219,91.268,418.897,171.051,33.329,156.251
C02727=1052.224,91.517,418.878,171.052,33.331,156.251
C02728=1052.231,91.767,418.859,171.054,33.333,156.252
C02729=1052.237,92.016,418.840,171.056,33.336,156.252
C02730=1052.243,92.265,418.821,171.057,33.338,156.252
C02731=1052.249,92.514,418.801,171.059,33.340,156.253
C02732=1052.255,92.763,418.783,171.061,33.342,156.253
C02733=1052.261,93.013,418.763,171.062,33.344,156.253
C02734=1052.268,93.262,418.745,171.064,33.346,156.254
C02735=1052.274,93.547,418.724,171.066,33.349,156.254
C02736=1052.281,93.832,418.702,171.068,33.351,156.255
C02737=1052.288,94.119,418.680,171.070,33.354,156.255
C02738=1052.295,94.404,418.658,171.071,33.356,156.255
C02739=1052.301,94.653,418.639,171.073,33.358,156.256
C02740=1052.307,94.902,418.620,171.075,33.361,156.256
C02741=1052.313,95.152,418.601,171.076,33.363,156.257
C02742=1052.319,95.400,418.581,171.078,33.365,156.257
C02743=1052.325,95.649,418.562,171.080,33.367,156.257
C02744=1052.332,95.899,418.544,171.081,33.369,156.258
C02745=1052.337,96.148,418.524,171.083,33.371,156.258
C02746=1052.344,96.397,418.506,171.085,33.374,156.258
C02747=1052.349,96.647,418.486,171.086,33.376,156.259
C02748=1052.356,96.895,418.467,171.088,33.378,156.259
C02749=1052.362,97.145,418.448,171.090,33.380,156.259
C02750=1052.368,97.394,418.429,171.091,33.382,156.260
C02751=1052.374,97.643,418.410,171.093,33.384,156.260
C02752=1052.380,97.893,418.391,171.095,33.387,156.261
C02753=1052.386,98.141,418.371,171.096,33.389,156.261
C02754=1052.392,98.390,418.352,171.098,33.391,156.261
C02755=1052.398,98.640,418.333,171.100,33.393,156.262
C02756=1052.405,98.890,418.314,171.101,33.395,156.262
C02757=1052.411,99.138,418.294,171.103,33.397,156.262
C02758=1052.417,99.388,418.275,171.104,33.400,156.263
C02759=1052.424,99.637,418.257,171.106,33.402,156.263
C02760=1052.429,99.886,418.237,171.108,33.404,156.263
C02761=1052.435,100.135,418.217,171.109,33.406,156.264
C02762=1052.442,100.384,418.199,171.111,33.408,156.264
C02763=1052.447,100.634,418.179,171.113,33.410,156.264
C02764=1052.454,100.882,418.160,171.114,33.413,156.265
C02765=1052.460,101.132,418.141,171.116,33.415,156.265
C02766=1052.465,101.381,418.122,171.118,33.417,156.265
C02767=1052.471,101.630,418.102,171.119,33.419,156.266
C02768=1052.478,101.880,418.082,171.121,33.421,156.266
C02769=1052.484,102.128,418.063,171.123,33.424,156.267
C02770=1052.490,102.378,418.043,171.124,33.426,156.267
C02771=1052.496,102.627,418.024,171.126,33.428,156.267
C02772=1052.502,102.876,418.004,171.128,33.430,156.268
C02773=1052.508,103.126,417.985,171.129,33.432,156.268
C02774=1052.514,103.374,417.966,171.131,33.435,156.269
C02775=1052.520,103.623,417.946,171.133,33.437,156.269
C02776=1052.526,103.873,417.927,171.135,33.439,156.269
C02777=1052.532,104.122,417.907,171.137,33.441,156.270
C02778=1052.537,104.371,417.888,171.139,33.443,156.270
C02779=1052.544,104.620,417.869,171.140,33.446,156.270
C02780=1052.550,104.870,417.849,171.142,33.448,156.271
C02781=1052.556,105.119,417.829,171.144,33.450,156.271
C02782=1052.562,105.368,417.810,171.145,33.452,156.271
C02783=1052.568,105.617,417.790,171.147,33.455,156.272
C02784=1052.574,105.866,417.771,171.149,33.457,156.272
C02785=1052.580,106.115,417.751,171.150,33.459,156.273
C02786=1052.586,106.364,417.732,171.152,33.461,156.273
C02787=1052.593,106.614,417.712,171.154,33.463,156.273
C02788=1052.598,106.863,417.692,171.155,33.466,156.274
C02789=1052.604,107.112,417.672,171.157,33.468,156.274
C02790=1052.611,107.360,417.653,171.159,33.470,156.274
C02791=1052.617,107.610,417.634,171.160,33.472,156.275
C02792=1052.623,107.859,417.614,171.162,33.474,156.275
C02793=1052.629,108.109,417.594,171.164,33.477,156.276
C02794=1052.635,108.358,417.574,171.165,33.479,156.276
C02795=1052.641,108.607,417.555,171.167,33.481,156.276
C02796=1052.647,108.856,417.535,171.169,33.483,156.277
C02797=1052.654,109.104,417.516,171.170,33.485,156.277
C02798=1052.660,109.355,417.496,171.172,33.487,156.277
C02799=1052.666,109.640,417.474,171.174,33.490,156.278
C02800=1052.674,109.925,417.450,171.176,33.493,156.278
C02801=1052.681,110.211,417.428,171.178,33.495,156.279
C02802=1052.687,110.496,417.406,171.180,33.498,156.279
C02803=1052.693,110.745,417.386,171.182,33.500,156.279
C02804=1052.699,110.995,417.366,171.183,33.502,156.280
C02805=1052.705,111.244,417.346,171.185,33.504,156.280
C02806=1052.711,111.492,417.326,171.187,33.506,156.280
C02807=1052.717,111.742,417.307,171.188,33.509,156.281
C02808=1052.724,111.991,417.286,171.190,33.511,156.281
C02809=1052.730,112.240,417.267,171.192,33.513,156.282
C02810=1052.736,112.489,417.247,171.193,33.515,156.282
C02811=1052.741,112.738,417.227,171.195,33.518,156.282
C02812=1052.747,112.987,417.207,171.197,33.520,156.283
C02813=1052.754,113.237,417.187,171.198,33.522,156.283
C02814=1052.760,113.486,417.167,171.200,33.524,156.283
C02815=1052.766,113.735,417.148,171.202,33.526,156.284
C02816=1052.772,113.984,417.128,171.203,33.529,156.284
C02817=1052.778,114.233,417.108,171.206,33.531,156.285
C02818=1052.784,114.482,417.088,171.208,33.533,156.285
C02819=1052.790,114.731,417.068,171.209,33.535,156.285
C02820=1052.795,114.981,417.048,171.211,33.538,156.286
C02821=1052.802,115.230,417.027,171.213,33.540,156.286
C02822=1052.808,115.479,417.008,171.215,33.542,156.286
C02823=1052.814,115.728,416.988,171.216,33.545,156.287
C02824=1052.819,115.977,416.967,171.218,33.547,156.287
C02825=1052.825,116.226,416.947,171.220,33.549,156.288
C02826=1052.832,116.475,416.927,171.221,33.551,156.288
C02827=1052.838,116.724,416.907,171.223,33.554,156.288
C02828=1052.843,116.973,416.886,171.225,33.556,156.289
C02829=1052.849,117.222,416.866,171.226,33.558,156.289
C02830=1052.855,117.472,416.847,171.228,33.560,156.290
C02831=1052.860,117.721,416.826,171.230,33.563,156.290
C02832=1052.866,117.970,416.806,171.231,33.565,156.290
C02833=1052.872,118.219,416.786,171.233,33.567,156.291
C02834=1052.879,118.469,416.766,171.235,33.570,156.291
C02835=1052.884,118.718,416.745,171.237,33.572,156.292
C02836=1052.890,118.966,416.725,171.238,33.574,156.292
C02837=1052.897,119.216,416.705,171.240,33.576,156.292
C02838=1052.903,119.465,416.685,171.242,33.579,156.293
C02839=1052.908,119.714,416.664,171.243,33.581,156.293
C02840=1052.915,119.963,416.644,171.245,33.583,156.293
C02841=1052.921,120.212,416.624,171.247,33.585,156.294
C02842=1052.926,120.461,416.604,171.248,33.588,156.294
C02843=1052.932,120.710,416.584,171.250,33.590,156.295
C02844=1052.939,120.960,416.563,171.252,33.592,156.295
C02845=1052.945,121.208,416.543,171.254,33.594,156.295
C02846=1052.950,121.457,416.522,171.255,33.597,156.296
C02847=1052.957,121.707,416.502,171.257,33.599,156.296
C02848=1052.963,121.955,416.482,171.260,33.601,156.297
C02849=1052.969,122.205,416.461,171.261,33.603,156.297
C02850=1052.975,122.454,416.441,171.263,33.606,156.297
C02851=1052.981,122.703,416.421,171.265,33.608,156.298
C02852=1052.986,122.953,416.400,171.267,33.610,156.298
C02853=1052.992,123.201,416.380,171.268,33.612,156.298
C02854=1052.998,123.450,416.360,171.270,33.615,156.299
C02855=1053.005,123.699,416.339,171.272,33.617,156.299
C02856=1053.011,123.948,416.319,171.274,33.619,156.300
C02857=1053.017,124.198,416.298,171.275,33.621,156.300
C02858=1053.022,124.447,416.278,171.277,33.624,156.300
C02859=1053.028,124.696,416.258,171.279,33.626,156.301
C02860=1053.035,124.945,416.237,171.281,33.628,156.301
C02861=1053.041,125.194,416.216,171.282,33.630,156.301
C02862=1053.047,125.443,416.196,171.284,33.633,156.302
C02863=1053.054,125.728,416.173,171.286,33.635,156.302
C02864=1053.060,126.014,416.150,171.288,33.637,156.303
C02865=1053.067,126.299,416.126,171.290,33.640,156.303
C02866=1053.074,126.585,416.102,171.292,33.643,156.304
C02867=1053.081,126.834,416.082,171.294,33.645,156.304
C02868=1053.087,127.082,416.061,171.295,33.647,156.304
C02869=1053.092,127.332,416.041,171.297,33.650,156.305
C02870=1053.099,127.581,416.020,171.299,33.652,156.305
C02871=1053.105,127.829,416.000,171.301,33.654,156.305
C02872=1053.111,128.079,415.979,171.302,33.656,156.306
C02873=1053.117,128.328,415.959,171.304,33.659,156.306
C02874=1053.124,128.577,415.939,171.306,33.661,156.307
C02875=1053.129,128.826,415.917,171.309,33.663,156.307
C02876=1053.136,129.075,415.897,171.311,33.665,156.307
C02877=1053.142,129.324,415.877,171.312,33.667,156.308
C02878=1053.148,129.573,415.855,171.314,33.670,156.308
C02879=1053.154,129.822,415.835,171.316,33.672,156.308
C02880=1053.160,130.072,415.814,171.318,33.674,156.309
C02881=1053.166,130.320,415.794,171.319,33.676,156.309
C02882=1053.173,130.570,415.773,171.321,33.679,156.310
C02883=1053.178,130.818,415.752,171.323,33.681,156.310
C02884=1053.185,131.068,415.732,171.325,33.683,156.310
C02885=1053.192,131.317,415.712,171.326,33.685,156.311
C02886=1053.197,131.566,415.690,171.328,33.687,156.311
C02887=1053.204,131.815,415.670,171.330,33.690,156.312
C02888=1053.209,132.064,415.649,171.332,33.692,156.312
C02889=1053.215,132.314,415.628,171.334,33.694,156.312
C02890=1053.221,132.562,415.607,171.335,33.697,156.313
C02891=1053.227,132.811,415.587,171.337,33.699,156.313
C02892=1053.233,133.060,415.565,171.339,33.701,156.313
C02893=1053.239,133.309,415.545,171.341,33.704,156.314
C02894=1053.245,133.558,415.523,171.342,33.706,156.314
C02895=1053.251,133.808,415.502,171.344,33.708,156.315
C02896=1053.257,134.056,415.482,171.346,33.710,156.315
C02897=1053.263,134.306,415.461,171.348,33.713,156.315
C02898=1053.269,134.555,415.440,171.349,33.715,156.316
C02899=1053.275,134.804,415.419,171.351,33.717,156.316
C02900=1053.281,135.053,415.398,171.354,33.720,156.317
C02901=1053.287,135.302,415.377,171.356,33.722,156.317
C02902=1053.293,135.551,415.356,171.358,33.724,156.317
C02903=1053.299,135.800,415.335,171.359,33.726,156.318
C02904=1053.304,136.049,415.314,171.361,33.729,156.318
C02905=1053.311,136.298,415.293,171.363,33.731,156.319
C02906=1053.316,136.547,415.273,171.365,33.733,156.319
C02907=1053.323,136.796,415.251,171.366,33.736,156.319
C02908=1053.330,137.045,415.230,171.368,33.738,156.320
C02909=1053.335,137.294,415.209,171.370,33.740,156.320
C02910=1053.341,137.543,415.188,171.372,33.742,156.321
C02911=1053.347,137.792,415.166,171.374,33.745,156.321
C02912=1053.353,138.041,415.146,171.375,33.747,156.321
C02913=1053.359,138.291,415.124,171.377,33.749,156.322
C02914=1053.365,138.539,415.103,171.379,33.752,156.322
C02915=1053.371,138.789,415.082,171.381,33.754,156.322
C02916=1053.377,139.037,415.062,171.383,33.756,156.323
C02917=1053.383,139.286,415.040,171.384,33.759,156.323
C02918=1053.389,139.536,415.018,171.386,33.761,156.324
C02919=1053.395,139.785,414.998,171.388,33.763,156.324
C02920=1053.401,140.034,414.977,171.390,33.765,156.324
C02921=1053.407,140.282,414.955,171.393,33.768,156.325
C02922=1053.413,140.531,414.934,171.394,33.770,156.325
C02923=1053.419,140.781,414.913,171.396,33.772,156.326
C02924=1053.425,141.030,414.892,171.398,33.775,156.326
C02925=1053.431,141.279,414.870,171.400,33.777,156.327
C02926=1053.436,141.527,414.849,171.402,33.779,156.327
C02927=1053.443,141.813,414.825,171.404,33.782,156.327
C02928=1053.451,142.098,414.800,171.406,33.785,156.328
C02929=1053.457,142.384,414.775,171.408,33.788,156.328
C02930=1053.464,142.669,414.751,171.410,33.790,156.329
C02931=1053.470,142.917,414.730,171.412,33.793,156.329
C02932=1053.476,143.167,414.708,171.414,33.795,156.330
C02933=1053.482,143.416,414.687,171.415,33.797,156.330
C02934=1053.488,143.664,414.665,171.417,33.800,156.330
C02935=1053.494,143.914,414.644,171.419,33.802,156.331
C02936=1053.500,144.163,414.622,171.421,33.804,156.331
C02937=1053.505,144.411,414.601,171.423,33.807,156.332
C02938=1053.511,144.661,414.580,171.425,33.809,156.332
C02939=1053.518,144.910,414.559,171.426,33.811,156.332
C02940=1053.524,145.158,414.538,171.429,33.814,156.333
C02941=1053.530,145.408,414.516,171.431,33.816,156.333
C02942=1053.536,145.657,414.494,171.433,33.818,156.334
C02943=1053.542,145.905,414.473,171.435,33.820,156.334
C02944=1053.548,146.155,414.451,171.437,33.823,156.334
C02945=1053.554,146.404,414.430,171.438,33.825,156.335
C02946=1053.560,146.653,414.408,171.440,33.827,156.335
C02947=1053.566,146.902,414.387,171.442,33.830,156.336
C02948=1053.572,147.151,414.365,171.444,33.832,156.336
C02949=1053.578,147.400,414.344,171.446,33.834,156.336
C02950=1053.584,147.649,414.322,171.448,33.837,156.337
C02951=1053.590,147.898,414.301,171.450,33.839,156.337
C02952=1053.596,148.147,414.279,171.451,33.841,156.338
C02953=1053.602,148.395,414.257,171.453,33.844,156.338
C02954=1053.608,148.644,414.235,171.455,33.846,156.338
C02955=1053.614,148.893,414.214,171.457,33.848,156.339
C02956=1053.620,149.143,414.192,171.459,33.851,156.339
C02957=1053.626,149.392,414.170,171.461,33.853,156.340
C02958=1053.631,149.640,414.149,171.463,33.856,156.340
C02959=1053.637,149.890,414.127,171.465,33.858,156.340
C02960=1053.644,150.139,414.105,171.467,33.860,156.341
C02961=1053.650,150.387,414.083,171.469,33.863,156.341
C02962=1053.656,150.636,414.062,171.471,33.865,156.342
C02963=1053.661,150.885,414.039,171.473,33.867,156.342
C02964=1053.667,151.135,414.018,171.475,33.870,156.343
C02965=1053.673,151.384,413.996,171.477,33.872,156.343
C02966=1053.679,151.632,413.975,171.478,33.874,156.343
C02967=1053.685,151.881,413.953,171.480,33.877,156.344
C02968=1053.691,152.130,413.930,171.482,33.879,156.344
C02969=1053.697,152.380,413.909,171.484,33.882,156.345
C02970=1053.703,152.629,413.887,171.486,33.884,156.345
C02971=1053.709,152.877,413.865,171.488,33.887,156.345
C02972=1053.715,153.126,413.843,171.490,33.889,156.346
C02973=1053.721,153.375,413.821,171.491,33.892,156.346
C02974=1053.727,153.625,413.800,171.493,33.893,156.347
C02975=1053.733,153.873,413.777,171.496,33.896,156.347
C02976=1053.739,154.122,413.756,171.498,33.899,156.348
C02977=1053.744,154.371,413.734,171.500,33.901,156.348
C02978=1053.751,154.620,413.711,171.502,33.903,156.348
C02979=1053.757,154.869,413.690,171.504,33.906,156.349
C02980=1053.763,155.118,413.668,171.506,33.908,156.349
C02981=1053.769,155.367,413.645,171.508,33.911,156.350
C02982=1053.774,155.616,413.624,171.509,33.913,156.350
C02983=1053.780,155.865,413.602,171.511,33.915,156.350
C02984=1053.786,156.114,413.579,171.513,33.918,156.351
C02985=1053.792,156.363,413.558,171.515,33.920,156.351
C02986=1053.799,156.612,413.535,171.517,33.923,156.352
C02987=1053.804,156.861,413.513,171.519,33.925,156.352
C02988=1053.810,157.109,413.491,171.521,33.927,156.353
C02989=1053.816,157.358,413.470,171.523,33.930,156.353
C02990=1053.822,157.608,413.447,171.525,33.932,156.353
C02991=1053.829,157.892,413.422,171.528,33.935,156.354
C02992=1053.836,158.178,413.396,171.530,33.937,156.354
C02993=1053.843,158.462,413.371,171.532,33.941,156.355
C02994=1053.849,158.747,413.346,171.534,33.943,156.355
C02995=1053.856,158.996,413.323,171.536,33.946,156.356
C02996=1053.862,159.245,413.302,171.538,33.948,156.356
C02997=1053.868,159.494,413.279,171.540,33.950,156.357
C02998=1053.874,159.743,413.257,171.542,33.953,156.357
C02999=1053.879,159.992,413.234,171.544,33.955,156.357
C03000=1053.885,160.241,413.213,171.546,33.958,156.358
C03001=1053.892,160.489,413.190,171.548,33.960,156.358
C03002=1053.897,160.739,413.168,171.550,33.962,156.359
C03003=1053.903,160.987,413.146,171.552,33.965,156.359
C03004=1053.909,161.236,413.123,171.554,33.967,156.360
C03005=1053.915,161.486,413.101,171.557,33.970,156.360
C03006=1053.920,161.735,413.078,171.559,33.972,156.360
C03007=1053.927,161.983,413.055,171.560,33.975,156.361
C03008=1053.932,162.232,413.034,171.562,33.977,156.361
C03009=1053.937,162.481,413.011,171.564,33.980,156.362
C03010=1053.943,162.730,412.988,171.566,33.982,156.362
C03011=1053.949,162.979,412.966,171.568,33.985,156.363
C03012=1053.955,163.228,412.943,171.570,33.988,156.363
C03013=1053.961,163.477,412.920,171.572,33.990,156.364
C03014=1053.966,163.726,412.897,171.574,33.993,156.364
C03015=1053.973,163.975,412.876,171.576,33.995,156.364
C03016=1053.978,164.224,412.853,171.578,33.998,156.365
C03017=1053.984,164.473,412.830,171.580,34.000,156.365
C03018=1053.989,164.721,412.807,171.583,34.003,156.366
C03019=1053.995,164.970,412.785,171.585,34.005,156.366
C03020=1054.001,165.219,412.763,171.586,34.008,156.367
C03021=1054.007,165.468,412.740,171.588,34.010,156.367
C03022=1054.013,165.717,412.717,171.590,34.013,156.368
C03023=1054.019,165.965,412.694,171.592,34.015,156.368
C03024=1054.024,166.215,412.672,171.594,34.018,156.369
C03025=1054.030,166.464,412.649,171.596,34.020,156.369
C03026=1054.036,166.713,412.626,171.598,34.023,156.369
C03027=1054.042,166.962,412.603,171.600,34.025,156.370
C03028=1054.048,167.210,412.581,171.602,34.028,156.370
C03029=1054.054,167.459,412.558,171.604,34.031,156.371
C03030=1054.060,167.708,412.535,171.606,34.033,156.371
C03031=1054.065,167.958,412.513,171.609,34.036,156.372
C03032=1054.071,168.206,412.490,171.611,34.038,156.372
C03033=1054.077,168.455,412.467,171.613,34.041,156.373
C03034=1054.083,168.704,412.444,171.615,34.043,156.373
C03035=1054.089,168.953,412.422,171.617,34.046,156.373
C03036=1054.094,169.202,412.399,171.619,34.048,156.374
C03037=1054.101,169.450,412.376,171.621,34.051,156.374
C03038=1054.107,169.699,412.353,171.623,34.053,156.375
C03039=1054.112,169.948,412.330,171.625,34.056,156.375
C03040=1054.118,170.197,412.307,171.627,34.058,156.376
C03041=1054.124,170.446,412.284,171.629,34.061,156.376
C03042=1054.130,170.695,412.262,171.631,34.063,156.377
C03043=1054.136,170.943,412.239,171.634,34.066,156.377
C03044=1054.142,171.192,412.216,171.636,34.069,156.377
C03045=1054.147,171.441,412.193,171.638,34.071,156.378
C03046=1054.154,171.691,412.170,171.640,34.074,156.378
C03047=1054.159,171.940,412.147,171.642,34.076,156.379
C03048=1054.166,172.188,412.125,171.644,34.079,156.379
C03049=1054.172,172.437,412.102,171.646,34.081,156.380
C03050=1054.177,172.686,412.079,171.648,34.084,156.380
C03051=1054.183,172.935,412.056,171.650,34.086,156.381
C03052=1054.189,173.184,412.033,171.652,34.089,156.381
C03053=1054.195,173.432,412.009,171.654,34.091,156.382
C03054=1054.201,173.681,411.987,171.656,34.094,156.382
C03055=1054.208,173.966,411.960,171.659,34.097,156.383
C03056=1054.215,174.251,411.935,171.662,34.100,156.383
C03057=1054.221,174.535,411.908,171.664,34.103,156.384
C03058=1054.228,174.819,411.882,171.666,34.105,156.384
C03059=1054.234,175.068,411.859,171.668,34.108,156.384
C03060=1054.241,175.317,411.835,171.670,34.110,156.385
C03061=1054.246,175.566,411.812,171.672,34.113,156.385
C03062=1054.252,175.815,411.789,171.674,34.115,156.386
C03063=1054.259,176.064,411.767,171.676,34.118,156.386
C03064=1054.264,176.312,411.744,171.678,34.120,156.387
C03065=1054.270,176.561,411.720,171.681,34.123,156.387
C03066=1054.277,176.810,411.697,171.683,34.125,156.388
C03067=1054.282,177.059,411.674,171.686,34.128,156.388
C03068=1054.288,177.308,411.651,171.688,34.130,156.388
C03069=1054.294,177.556,411.627,171.690,34.133,156.389
C03070=1054.301,177.806,411.604,171.692,34.136,156.389
C03071=1054.306,178.055,411.581,171.694,34.138,156.390
C03072=1054.313,178.303,411.558,171.696,34.141,156.390
C03073=1054.319,178.552,411.535,171.698,34.143,156.391
C03074=1054.325,178.801,411.512,171.700,34.146,156.391
C03075=1054.331,179.050,411.489,171.702,34.149,156.392
C03076=1054.337,179.298,411.465,171.704,34.151,156.392
C03077=1054.343,179.547,411.442,171.706,34.154,156.393
C03078=1054.349,179.796,411.418,171.709,34.156,156.393
C03079=1054.355,180.045,411.395,171.712,34.159,156.394
C03080=1054.361,180.294,411.372,171.714,34.161,156.394
C03081=1054.367,180.542,411.348,171.716,34.164,156.394
C03082=1054.374,180.792,411.326,171.718,34.166,156.395
C03083=1054.380,181.041,411.303,171.720,34.169,156.395
C03084=1054.386,181.289,411.279,171.722,34.171,156.396
C03085=1054.392,181.538,411.256,171.724,34.174,156.396
C03086=1054.398,181.787,411.232,171.726,34.176,156.397
C03087=1054.404,182.036,411.209,171.728,34.179,156.397
C03088=1054.410,182.285,411.185,171.730,34.182,156.398
C03089=1054.416,182.534,411.162,171.734,34.184,156.398
C03090=1054.422,182.782,411.139,171.736,34.187,156.399
C03091=1054.428,183.031,411.115,171.738,34.189,156.399
C03092=1054.435,183.280,411.092,171.740,34.192,156.399
C03093=1054.440,183.529,411.069,171.742,34.194,156.400
C03094=1054.447,183.778,411.045,171.744,34.197,156.400
C03095=1054.453,184.026,411.022,171.746,34.199,156.401
C03096=1054.459,184.275,410.998,171.748,34.202,156.401
C03097=1054.465,184.524,410.975,171.750,34.204,156.402
C03098=1054.471,184.773,410.951,171.753,34.207,156.402
C03099=1054.476,185.022,410.928,171.756,34.210,156.403
C03100=1054.483,185.271,410.904,171.758,34.212,156.403
C03101=1054.488,185.519,410.879,171.760,34.216,156.404
C03102=1054.494,185.768,410.856,171.762,34.218,156.404
C03103=1054.499,186.017,410.832,171.764,34.221,156.405
C03104=1054.506,186.266,410.808,171.766,34.224,156.405
C03105=1054.511,186.514,410.784,171.768,34.226,156.406
C03106=1054.517,186.763,410.761,171.770,34.229,156.406
C03107=1054.523,187.012,410.737,171.773,34.232,156.407
C03108=1054.529,187.261,410.713,171.775,34.234,156.407
C03109=1054.535,187.509,410.689,171.778,34.237,156.408
C03110=1054.540,187.759,410.665,171.780,34.240,156.408
C03111=1054.546,188.007,410.641,171.782,34.243,156.409
C03112=1054.552,188.256,410.617,171.784,34.245,156.409
C03113=1054.558,188.505,410.593,171.786,34.248,156.410
C03114=1054.563,188.754,410.569,171.788,34.251,156.410
C03115=1054.569,189.002,410.546,171.791,34.254,156.411
C03116=1054.576,189.251,410.522,171.793,34.256,156.411
C03117=1054.581,189.500,410.498,171.795,34.259,156.412
C03118=1054.587,189.748,410.474,171.798,34.262,156.412
C03119=1054.594,190.033,410.447,171.800,34.265,156.413
C03120=1054.601,190.317,410.419,171.803,34.268,156.413
C03121=1054.607,190.601,410.391,171.805,34.271,156.414
C03122=1054.613,190.885,410.364,171.808,34.274,156.414
C03123=1054.620,191.134,410.340,171.810,34.277,156.415
C03124=1054.625,191.383,410.316,171.812,34.279,156.415
C03125=1054.632,191.632,410.292,171.814,34.283,156.416
C03126=1054.637,191.880,410.268,171.816,34.285,156.416
C03127=1054.644,192.129,410.244,171.820,34.288,156.417
C03128=1054.649,192.378,410.219,171.822,34.291,156.417
C03129=1054.655,192.626,410.196,171.824,34.293,156.418
C03130=1054.661,192.875,410.171,171.826,34.296,156.418
C03131=1054.667,193.124,410.147,171.828,34.299,156.419
C03132=1054.673,193.373,410.123,171.830,34.301,156.419
C03133=1054.679,193.621,410.099,171.833,34.305,156.420
C03134=1054.685,193.871,410.075,171.835,34.307,156.420
C03135=1054.691,194.119,410.051,171.838,34.310,156.421
C03136=1054.697,194.368,410.026,171.840,34.313,156.421
C03137=1054.703,194.616,410.003,171.842,34.315,156.422
C03138=1054.709,194.866,409.978,171.845,34.318,156.422
C03139=1054.715,195.114,409.954,171.847,34.321,156.423
C03140=1054.721,195.363,409.930,171.849,34.323,156.423
C03141=1054.727,195.612,409.906,171.851,34.326,156.424
C03142=1054.733,195.860,409.881,171.853,34.329,156.424
C03143=1054.739,196.109,409.857,171.856,34.332,156.425
C03144=1054.745,196.358,409.832,171.859,34.335,156.425
C03145=1054.751,196.606,409.809,171.861,34.337,156.426
C03146=1054.757,196.855,409.784,171.863,34.340,156.426
C03147=1054.763,197.104,409.760,171.866,34.343,156.427
C03148=1054.769,197.353,409.736,171.868,34.346,156.427
C03149=1054.775,197.602,409.711,171.870,34.348,156.428
C03150=1054.781,197.850,409.687,171.872,34.351,156.428
C03151=1054.787,198.099,409.662,171.875,34.354,156.429
C03152=1054.793,198.347,409.639,171.877,34.356,156.429
C03153=1054.799,198.597,409.614,171.880,34.360,156.430
C03154=1054.806,198.845,409.589,171.882,34.362,156.430
C03155=1054.811,199.094,409.565,171.884,34.365,156.431
C03156=1054.817,199.343,409.540,171.887,34.368,156.431
C03157=1054.823,199.591,409.517,171.889,34.371,156.432
C03158=1054.829,199.840,409.491,171.891,34.373,156.432
C03159=1054.836,200.089,409.467,171.894,34.376,156.433
C03160=1054.841,200.337,409.443,171.896,34.379,156.433
C03161=1054.848,200.586,409.418,171.899,34.381,156.434
C03162=1054.854,200.835,409.394,171.901,34.385,156.434
C03163=1054.859,201.084,409.369,171.904,34.387,156.435
C03164=1054.866,201.332,409.345,171.906,34.390,156.435
C03165=1054.872,201.581,409.320,171.908,34.393,156.436
C03166=1054.878,201.830,409.296,171.910,34.396,156.437
C03167=1054.884,202.078,409.271,171.913,34.398,156.437
C03168=1054.890,202.328,409.246,171.915,34.401,156.438
C03169=1054.896,202.576,409.221,171.918,34.404,156.438
C03170=1054.902,202.825,409.197,171.920,34.407,156.439
C03171=1054.907,203.073,409.172,171.923,34.410,156.439
C03172=1054.913,203.322,409.147,171.925,34.413,156.440
C03173=1054.919,203.571,409.122,171.927,34.416,156.440
C03174=1054.925,203.819,409.098,171.930,34.419,156.441
C03175=1054.932,204.068,409.073,171.932,34.421,156.441
C03176=1054.938,204.317,409.048,171.935,34.424,156.442
C03177=1054.943,204.565,409.023,171.937,34.428,156.442
C03178=1054.949,204.814,408.999,171.940,34.430,156.443
C03179=1054.955,205.063,408.973,171.942,34.433,156.443
C03180=1054.961,205.312,408.949,171.944,34.436,156.444
C03181=1054.967,205.560,408.924,171.947,34.439,156.444
C03182=1054.973,205.809,408.898,171.949,34.442,156.445
C03183=1054.998,206.860,408.793,172.155,34.534,156.459
C03184=1055.004,207.101,408.768,172.157,34.537,156.460
C03185=1055.011,207.341,408.744,172.159,34.541,156.461
C03186=1055.017,207.581,408.719,172.161,34.544,156.461
C03187=1055.022,207.823,408.694,172.162,34.548,156.462
C03188=1055.029,208.063,408.669,172.164,34.552,156.463
C03189=1055.035,208.303,408.644,172.167,34.555,156.463
C03190=1055.041,208.544,408.618,172.168,34.559,156.464
C03191=1055.047,208.784,408.593,172.170,34.562,156.465
C03192=1055.054,209.032,408.567,172.172,34.566,156.466
C03193=1055.059,209.281,408.541,172.174,34.570,156.466
C03194=1055.066,209.530,408.515,172.176,34.573,156.467
C03195=1055.072,209.779,408.490,172.178,34.577,156.468
C03196=1055.079,210.027,408.464,172.180,34.581,156.468
C03197=1055.084,210.276,408.438,172.182,34.584,156.469
C03198=1055.091,210.524,408.412,172.184,34.589,156.470
C03199=1055.098,210.773,408.386,172.186,34.592,156.471
C03200=1055.104,211.021,408.359,172.188,34.596,156.471
C03201=1055.110,211.270,408.333,172.190,34.599,156.472
C03202=1055.116,211.519,408.307,172.192,34.603,156.473
C03203=1055.123,211.767,408.281,172.194,34.607,156.474
C03204=1055.129,212.015,408.255,172.196,34.611,156.474
C03205=1055.135,212.264,408.229,172.198,34.615,156.475
C03206=1055.141,212.512,408.203,172.200,34.618,156.476
C03207=1055.147,212.761,408.176,172.201,34.622,156.476
C03208=1055.154,213.010,408.151,172.204,34.625,156.477
C03209=1055.159,213.258,408.124,172.206,34.629,156.478
C03210=1055.166,213.506,408.098,172.208,34.633,156.479
C03211=1055.172,213.756,408.071,172.210,34.637,156.479
C03212=1055.179,214.004,408.045,172.212,34.641,156.480
C03213=1055.184,214.253,408.019,172.214,34.644,156.481
C03214=1055.191,214.501,407.993,172.216,34.648,156.482
C03215=1055.197,214.750,407.966,172.218,34.651,156.482
C03216=1055.203,214.998,407.940,172.220,34.656,156.483
C03217=1055.209,215.247,407.914,172.222,34.659,156.484
C03218=1055.216,215.495,407.887,172.224,34.663,156.485
C03219=1055.222,215.744,407.861,172.226,34.667,156.485
C03220=1055.229,215.992,407.835,172.228,34.670,156.486
C03221=1055.235,216.241,407.808,172.230,34.674,156.487
C03222=1055.241,216.490,407.782,172.232,34.677,156.487
C03223=1055.247,216.738,407.756,172.234,34.681,156.488
C03224=1055.253,216.987,407.729,172.236,34.685,156.489
C03225=1055.260,217.235,407.703,172.238,34.689,156.490
C03226=1055.266,217.483,407.676,172.241,34.693,156.490
C03227=1055.273,217.732,407.649,172.243,34.696,156.491
C03228=1055.279,217.981,407.623,172.245,34.700,156.492
C03229=1055.285,218.229,407.597,172.246,34.703,156.492
C03230=1055.291,218.478,407.570,172.248,34.707,156.493
C03231=1055.298,218.726,407.544,172.251,34.711,156.494
C03232=1055.304,218.975,407.517,172.253,34.714,156.495
C03233=1055.310,219.223,407.490,172.255,34.718,156.495
C03234=1055.317,219.471,407.464,172.257,34.721,156.496
C03235=1055.323,219.720,407.437,172.259,34.725,156.497
C03236=1055.329,219.968,407.411,172.261,34.729,156.497
C03237=1055.336,220.217,407.384,172.263,34.732,156.498
C03238=1055.342,220.466,407.357,172.265,34.736,156.499
C03239=1055.349,220.714,407.331,172.267,34.740,156.500
C03240=1055.355,220.957,407.305,172.270,34.743,156.500
C03241=1055.360,221.200,407.279,172.272,34.747,156.501
C03242=1055.366,221.443,407.252,172.273,34.750,156.502
C03243=1055.373,221.687,407.227,172.275,34.754,156.502
C03244=1055.379,221.930,407.200,172.278,34.758,156.503
C03245=1055.385,222.173,407.174,172.280,34.761,156.504
C03246=1055.391,222.417,407.148,172.282,34.765,156.505
C03247=1055.397,222.660,407.122,172.284,34.769,156.505
C03248=1055.403,222.908,407.095,172.286,34.772,156.506
C03249=1055.409,223.157,407.068,172.288,34.776,156.507
C03250=1055.416,223.404,407.041,172.290,34.779,156.507
C03251=1055.422,223.653,407.014,172.292,34.784,156.508
C03252=1055.428,223.902,406.988,172.294,34.787,156.509
C03253=1055.434,224.150,406.961,172.297,34.791,156.510
C03254=1055.440,224.399,406.933,172.299,34.794,156.510
C03255=1055.446,224.647,406.907,172.301,34.798,156.511
C03256=1055.453,224.896,406.880,172.303,34.802,156.512
C03257=1055.459,225.144,406.853,172.306,34.805,156.513
C03258=1055.466,225.393,406.826,172.307,34.809,156.513
C03259=1055.472,225.641,406.799,172.309,34.812,156.514
C03260=1055.478,225.890,406.772,172.311,34.816,156.515
C03261=1055.484,226.138,406.745,172.314,34.820,156.515
C03262=1055.491,226.386,406.718,172.316,34.823,156.516
C03263=1055.497,226.635,406.692,172.318,34.827,156.517
C03264=1055.504,226.883,406.664,172.320,34.831,156.518
C03265=1055.509,227.132,406.637,172.323,34.834,156.518
C03266=1055.516,227.381,406.610,172.325,34.838,156.519
C03267=1055.522,227.629,406.582,172.327,34.841,156.520
C03268=1055.528,227.877,406.556,172.329,34.845,156.520
C03269=1055.535,228.127,406.529,172.331,34.849,156.521
C03270=1055.541,228.374,406.502,172.334,34.852,156.522
C03271=1055.548,228.623,406.475,172.336,34.856,156.523
C03272=1055.554,228.871,406.448,172.338,34.860,156.523
C03273=1055.560,229.120,406.421,172.340,34.863,156.524
C03274=1055.567,229.368,406.393,172.343,34.867,156.525
C03275=1055.573,229.617,406.366,172.344,34.870,156.525
C03276=1055.579,229.865,406.339,172.346,34.874,156.526
C03277=1055.585,230.113,406.312,172.348,34.878,156.527
C03278=1055.592,230.362,406.284,172.351,34.881,156.528
C03279=1055.598,230.610,406.258,172.353,34.885,156.528
C03280=1055.604,230.859,406.229,172.355,34.888,156.529
C03281=1055.610,231.108,406.202,172.357,34.892,156.530
C03282=1055.616,231.356,406.175,172.360,34.896,156.530
C03283=1055.623,231.604,406.147,172.362,34.899,156.531
C03284=1055.628,231.853,406.120,172.364,34.903,156.532
C03285=1055.635,232.101,406.093,172.366,34.906,156.533
C03286=1055.642,232.350,406.066,172.369,34.910,156.533
C03287=1055.648,232.598,406.038,172.371,34.914,156.534
C03288=1055.654,232.846,406.011,172.373,34.917,156.535
C03289=1055.660,233.096,405.983,172.375,34.921,156.535
C03290=1055.666,233.343,405.956,172.378,34.925,156.536
C03291=1055.673,233.592,405.928,172.380,34.929,156.537
C03292=1055.678,233.840,405.901,172.382,34.932,156.538
C03293=1055.685,234.089,405.874,172.384,34.936,156.538
C03294=1055.691,234.337,405.845,172.387,34.939,156.539
C03295=1055.697,234.585,405.818,172.389,34.943,156.540
C03296=1055.703,234.825,405.792,172.391,34.947,156.541
C03297=1055.709,235.064,405.765,172.393,34.950,156.541
C03298=1055.715,235.303,405.738,172.396,34.953,156.542
C03299=1055.721,235.543,405.711,172.398,34.957,156.543
C03300=1055.727,235.781,405.686,172.400,34.961,156.543
C03301=1055.734,236.021,405.659,172.402,34.964,156.544
C03302=1055.740,236.260,405.632,172.405,34.967,156.545
C03303=1055.745,236.499,405.605,172.407,34.971,156.545
C03304=1055.752,236.747,405.578,172.409,34.974,156.546
C03305=1055.758,236.997,405.550,172.411,34.978,156.547
C03306=1055.764,237.244,405.523,172.414,34.982,156.548
C03307=1055.771,237.493,405.495,172.416,34.985,156.548
C03308=1055.776,237.742,405.467,172.418,34.989,156.549
C03309=1055.783,237.990,405.439,172.420,34.992,156.550
C03310=1055.789,238.238,405.411,172.423,34.996,156.550
C03311=1055.796,238.486,405.384,172.425,35.000,156.551
C03312=1055.802,238.735,405.355,172.427,35.003,156.552
C03313=1055.809,238.983,405.328,172.429,35.007,156.553
C03314=1055.815,239.231,405.300,172.432,35.010,156.553
C03315=1055.821,239.480,405.272,172.434,35.014,156.554
C03316=1055.827,239.728,405.244,172.436,35.018,156.555
C03317=1055.834,239.977,405.217,172.438,35.021,156.555
C03318=1055.839,240.225,405.189,172.441,35.025,156.556
C03319=1055.846,240.473,405.161,172.443,35.028,156.557
C03320=1055.853,240.722,405.133,172.445,35.032,156.558
C03321=1055.859,240.971,405.105,172.448,35.036,156.558
C03322=1055.865,241.219,405.077,172.451,35.039,156.559
C03323=1055.871,241.467,405.050,172.453,35.043,156.560
C03324=1055.877,241.715,405.021,172.455,35.046,156.561
C03325=1055.884,241.964,404.994,172.458,35.050,156.561
C03326=1055.890,242.213,404.965,172.460,35.054,156.562
C03327=1055.897,242.461,404.938,172.462,35.057,156.563
C03328=1055.902,242.709,404.909,172.464,35.061,156.563
C03329=1055.909,242.957,404.881,172.467,35.064,156.564
C03330=1055.915,243.206,404.853,172.469,35.068,156.565
C03331=1055.921,243.454,404.825,172.471,35.072,156.566
C03332=1055.927,243.703,404.797,172.473,35.075,156.566
C03333=1055.933,243.950,404.768,172.477,35.079,156.567
C03334=1055.940,244.199,404.740,172.479,35.082,156.568
C03335=1055.946,244.448,404.712,172.481,35.086,156.568
C03336=1055.952,244.696,404.684,172.483,35.090,156.569
C03337=1055.959,244.944,404.655,172.486,35.093,156.570
C03338=1055.965,245.193,404.627,172.488,35.097,156.571
C03339=1055.971,245.441,404.600,172.490,35.100,156.571
C03340=1055.977,245.689,404.571,172.493,35.104,156.572
C03341=1055.984,245.937,404.543,172.496,35.107,156.573
C03342=1055.990,246.186,404.515,172.498,35.111,156.573
C03343=1055.996,246.434,404.485,172.500,35.115,156.574
C03344=1056.002,246.683,404.457,172.503,35.118,156.575
C03345=1056.008,246.931,404.429,172.505,35.122,156.576
C03346=1056.014,247.179,404.401,172.507,35.125,156.576
C03347=1056.020,247.427,404.372,172.509,35.129,156.577
C03348=1056.026,247.676,404.343,172.512,35.133,156.578
C03349=1056.032,247.924,404.315,172.514,35.137,156.579
C03350=1056.038,248.172,404.286,172.517,35.140,156.579
C03351=1056.045,248.421,404.258,172.520,35.144,156.580
C03352=1056.050,248.657,404.231,172.522,35.147,156.581
C03353=1056.057,248.893,404.204,172.524,35.151,156.581
C03354=1056.062,249.130,404.176,172.526,35.154,156.582
C03355=1056.068,249.366,404.150,172.529,35.158,156.583
C03356=1056.074,249.602,404.123,172.531,35.161,156.584
C03357=1056.080,249.838,404.095,172.533,35.164,156.584
C03358=1056.086,250.074,404.068,172.535,35.168,156.585
C03359=1056.092,250.311,404.041,172.538,35.171,156.586
C03360=1056.097,250.558,404.012,172.540,35.175,156.586
C03361=1056.104,250.807,403.984,172.542,35.179,156.587
C03362=1056.110,251.055,403.955,172.546,35.182,156.588
C03363=1056.116,251.303,403.926,172.548,35.186,156.589
C03364=1056.122,251.552,403.898,172.550,35.189,156.589
C03365=1056.129,251.800,403.869,172.552,35.193,156.590
C03366=1056.135,252.048,403.840,172.555,35.197,156.591
C03367=1056.141,252.297,403.811,172.558,35.200,156.591
C03368=1056.147,252.545,403.782,172.560,35.204,156.592
C03369=1056.154,252.793,403.754,172.563,35.207,156.593
C03370=1056.160,253.042,403.726,172.565,35.211,156.594
C03371=1056.166,253.290,403.696,172.567,35.214,156.594
C03372=1056.172,253.538,403.667,172.570,35.218,156.595
C03373=1056.179,253.786,403.638,172.573,35.222,156.596
C03374=1056.185,254.035,403.610,172.575,35.225,156.597
C03375=1056.191,254.283,403.581,172.577,35.229,156.597
C03376=1056.197,254.531,403.552,172.580,35.232,156.598
C03377=1056.203,254.779,403.523,172.583,35.236,156.599
C03378=1056.210,255.027,403.495,172.585,35.240,156.599
C03379=1056.216,255.276,403.466,172.587,35.243,156.600
C03380=1056.223,255.525,403.437,172.590,35.247,156.601
C03381=1056.229,255.773,403.408,172.593,35.250,156.602
C03382=1056.236,256.021,403.379,172.595,35.254,156.602
C03383=1056.242,256.269,403.350,172.598,35.257,156.603
C03384=1056.248,256.517,403.321,172.600,35.261,156.604
C03385=1056.254,256.765,403.292,172.603,35.265,156.605
C03386=1056.260,257.014,403.263,172.605,35.268,156.605
C03387=1056.267,257.262,403.234,172.608,35.272,156.606
C03388=1056.273,257.510,403.205,172.610,35.275,156.607
C03389=1056.280,257.758,403.177,172.613,35.279,156.607
C03390=1056.287,258.007,403.147,172.616,35.282,156.608
C03391=1056.293,258.255,403.118,172.618,35.286,156.609
C03392=1056.299,258.503,403.089,172.620,35.290,156.610
C03393=1056.305,258.751,403.060,172.624,35.293,156.610
C03394=1056.312,258.999,403.031,172.626,35.297,156.611
C03395=1056.318,259.248,403.002,172.628,35.300,156.612
C03396=1056.325,259.496,402.973,172.631,35.304,156.613
C03397=1056.331,259.745,402.944,172.634,35.308,156.613
C03398=1056.337,259.993,402.915,172.636,35.311,156.614
C03399=1056.344,260.241,402.886,172.638,35.315,156.615
C03400=1056.350,260.489,402.857,172.642,35.318,156.615
C03401=1056.357,260.738,402.827,172.644,35.321,156.616
C03402=1056.363,260.985,402.797,172.646,35.325,156.617
C03403=1056.369,261.233,402.768,172.649,35.328,156.618
C03404=1056.376,261.482,402.739,172.652,35.332,156.618
C03405=1056.382,261.730,402.710,172.654,35.335,156.619
C03406=1056.389,261.979,402.681,172.657,35.339,156.620
C03407=1056.395,262.227,402.652,172.660,35.343,156.620
C03408=1056.401,262.462,402.624,172.662,35.346,156.621
C03409=1056.408,262.697,402.597,172.664,35.349,156.622
C03410=1056.414,262.932,402.569,172.668,35.353,156.623
C03411=1056.420,263.167,402.541,172.670,35.356,156.623
C03412=1056.426,263.402,402.513,172.672,35.359,156.624
C03413=1056.432,263.638,402.485,172.674,35.363,156.625
C03414=1056.438,263.873,402.457,172.677,35.366,156.625
C03415=1056.444,264.108,402.429,172.680,35.370,156.626
C03416=1056.450,264.356,402.400,172.682,35.374,156.627
C03417=1056.456,264.605,402.370,172.685,35.377,156.628
C03418=1056.462,264.853,402.340,172.688,35.381,156.628
C03419=1056.469,265.101,402.311,172.690,35.384,156.629
C03420=1056.474,265.349,402.281,172.693,35.388,156.630
C03421=1056.481,265.598,402.251,172.696,35.391,156.630
C03422=1056.488,265.846,402.222,172.698,35.395,156.631
C03423=1056.493,266.094,402.192,172.700,35.399,156.632
C03424=1056.500,266.342,402.163,172.704,35.402,156.633
C03425=1056.507,266.590,402.132,172.706,35.406,156.633
C03426=1056.512,266.838,402.103,172.708,35.409,156.634
C03427=1056.519,267.086,402.073,172.712,35.413,156.635
C03428=1056.526,267.335,402.044,172.714,35.417,156.636
C03429=1056.532,267.583,402.013,172.716,35.420,156.636
C03430=1056.538,267.831,401.984,172.720,35.424,156.637
C03431=1056.545,268.079,401.954,172.722,35.428,156.638
C03432=1056.550,268.327,401.925,172.725,35.431,156.639
C03433=1056.557,268.575,401.895,172.728,35.435,156.639
C03434=1056.563,268.823,401.865,172.730,35.438,156.640
C03435=1056.570,269.072,401.835,172.733,35.442,156.641
C03436=1056.576,269.320,401.806,172.736,35.445,156.642
C03437=1056.582,269.567,401.776,172.738,35.449,156.642
C03438=1056.589,269.816,401.746,172.741,35.453,156.643
C03439=1056.594,270.064,401.716,172.744,35.457,156.644
C03440=1056.602,270.312,401.686,172.747,35.460,156.645
C03441=1056.607,270.560,401.655,172.749,35.464,156.645
C03442=1056.614,270.808,401.626,172.752,35.467,156.646
C03443=1056.620,271.057,401.596,172.755,35.471,156.647
C03444=1056.627,271.304,401.566,172.757,35.474,156.648
C03445=1056.632,271.552,401.536,172.761,35.478,156.648
C03446=1056.639,271.801,401.506,172.763,35.482,156.649
C03447=1056.645,272.049,401.476,172.765,35.486,156.650
C03448=1056.652,272.297,401.445,172.769,35.489,156.651
C03449=1056.658,272.545,401.415,172.771,35.493,156.651
C03450=1056.664,272.793,401.386,172.774,35.496,156.652
C03451=1056.671,273.042,401.356,172.777,35.500,156.653
C03452=1056.677,273.289,401.325,172.780,35.503,156.654
C03453=1056.683,273.538,401.294,172.782,35.507,156.654
C03454=1056.690,273.785,401.265,172.785,35.511,156.655
C03455=1056.695,274.033,401.234,172.788,35.515,156.656
C03456=1056.702,274.282,401.204,172.790,35.518,156.657
C03457=1056.708,274.529,401.174,172.794,35.522,156.657
C03458=1056.715,274.778,401.143,172.796,35.525,156.658
C03459=1056.721,275.026,401.113,172.799,35.529,156.659
C03460=1056.727,275.274,401.083,172.802,35.533,156.660
C03461=1056.733,275.522,401.053,172.805,35.537,156.660
C03462=1056.740,275.771,401.022,172.807,35.540,156.661
C03463=1056.746,276.018,400.993,172.811,35.544,156.662
C03464=1056.752,276.255,400.963,172.813,35.547,156.663
C03465=1056.758,276.492,400.934,172.815,35.551,156.663
C03466=1056.764,276.730,400.905,172.819,35.554,156.664
C03467=1056.771,276.967,400.876,172.821,35.558,156.665
C03468=1056.777,277.204,400.846,172.823,35.561,156.666
C03469=1056.782,277.442,400.818,172.827,35.565,156.666
C03470=1056.788,277.679,400.788,172.829,35.568,156.667
C03471=1056.795,277.916,400.760,172.831,35.572,156.668
C03472=1056.801,278.164,400.729,172.835,35.576,156.669
C03473=1056.807,278.412,400.698,172.837,35.579,156.669
C03474=1056.814,278.660,400.667,172.840,35.583,156.670
C03475=1056.820,278.908,400.637,172.843,35.586,156.671
C03476=1056.827,279.156,400.607,172.846,35.590,156.672
C03477=1056.832,279.404,400.576,172.848,35.594,156.672
C03478=1056.839,279.652,400.545,172.852,35.597,156.673
C03479=1056.845,279.901,400.515,172.854,35.601,156.674
C03480=1056.851,280.148,400.484,172.857,35.604,156.675
C03481=1056.858,280.397,400.453,172.860,35.609,156.675
C03482=1056.864,280.644,400.423,172.863,35.612,156.676
C03483=1056.870,280.892,400.391,172.865,35.616,156.677
C03484=1056.877,281.140,400.361,172.869,35.620,156.678
C03485=1056.883,281.388,400.331,172.872,35.623,156.679
C03486=1056.889,281.636,400.300,172.874,35.627,156.679
C03487=1056.896,281.884,400.269,172.878,35.631,156.680
C03488=1056.902,282.133,400.238,172.880,35.634,156.681
C03489=1056.908,282.380,400.207,172.884,35.638,156.682
C03490=1056.915,282.628,400.176,172.886,35.642,156.682
C03491=1056.921,282.876,400.145,172.889,35.646,156.683
C03492=1056.927,283.124,400.115,172.892,35.649,156.684
C03493=1056.934,283.372,400.083,172.895,35.653,156.685
C03494=1056.939,283.620,400.052,172.897,35.657,156.686
C03495=1056.946,283.868,400.021,172.901,35.660,156.686
C03496=1056.952,284.117,399.990,172.903,35.664,156.687
C03497=1056.958,284.364,399.959,172.906,35.668,156.688
C03498=1056.965,284.612,399.928,172.910,35.672,156.689
C03499=1056.972,284.860,399.897,172.912,35.675,156.689
C03500=1056.977,285.108,399.867,172.916,35.679,156.690
C03501=1056.984,285.356,399.835,172.918,35.683,156.691
C03502=1056.990,285.604,399.804,172.921,35.686,156.692
C03503=1056.997,285.852,399.773,172.924,35.690,156.693
C03504=1057.003,286.100,399.743,172.927,35.694,156.693
C03505=1057.010,286.348,399.711,172.930,35.697,156.694
C03506=1057.016,286.595,399.680,172.933,35.701,156.695
C03507=1057.022,286.844,399.649,172.936,35.705,156.696
C03508=1057.029,287.092,399.618,172.938,35.709,156.696
C03509=1057.036,287.340,399.587,172.942,35.712,156.697
C03510=1057.042,287.587,399.556,172.945,35.716,156.698
C03511=1057.048,287.835,399.525,172.948,35.720,156.699
C03512=1057.055,288.083,399.493,172.951,35.723,156.700
C03513=1057.062,288.331,399.462,172.953,35.727,156.700
C03514=1057.067,288.579,399.431,172.957,35.731,156.701
C03515=1057.074,288.827,399.400,172.960,35.734,156.702
C03516=1057.080,289.075,399.368,172.962,35.739,156.703
C03517=1057.087,289.323,399.337,172.966,35.742,156.704
C03518=1057.092,289.570,399.305,172.969,35.746,156.704
C03519=1057.099,289.819,399.274,172.972,35.750,156.705
C03520=1057.106,290.062,399.243,172.975,35.753,156.706
C03521=1057.112,290.304,399.212,172.977,35.757,156.707
C03522=1057.117,290.547,399.182,172.981,35.761,156.708
C03523=1057.124,290.789,399.151,172.984,35.764,156.708
C03524=1057.131,291.032,399.120,172.987,35.768,156.709
C03525=1057.137,291.275,399.089,172.990,35.772,156.710
C03526=1057.143,291.518,399.058,172.992,35.775,156.711
C03527=1057.149,291.760,399.027,172.996,35.780,156.711
C03528=1057.155,292.008,398.996,172.999,35.783,156.712
C03529=1057.162,292.256,398.964,173.001,35.787,156.713
C03530=1057.168,292.504,398.932,173.005,35.791,156.714
C03531=1057.175,292.752,398.901,173.008,35.794,156.715
C03532=1057.181,293.000,398.870,173.011,35.798,156.715
C03533=1057.187,293.247,398.838,173.014,35.802,156.716
C03534=1057.194,293.495,398.806,173.017,35.806,156.717
C03535=1057.200,293.743,398.775,173.020,35.809,156.718
C03536=1057.206,293.991,398.743,173.023,35.813,156.719
C03537=1057.213,294.239,398.711,173.027,35.817,156.719
C03538=1057.219,294.487,398.679,173.029,35.821,156.720
C03539=1057.226,294.735,398.647,173.032,35.825,156.721
C03540=1057.233,294.983,398.616,173.036,35.829,156.722
C03541=1057.238,295.230,398.584,173.038,35.832,156.723
C03542=1057.245,295.478,398.553,173.042,35.836,156.724
C03543=1057.251,295.726,398.520,173.045,35.840,156.724
C03544=1057.258,295.974,398.489,173.048,35.844,156.725
C03545=1057.264,296.222,398.457,173.051,35.848,156.726
C03546=1057.271,296.470,398.425,173.054,35.851,156.727
C03547=1057.277,296.717,398.392,173.058,35.856,156.728
C03548=1057.283,296.966,398.360,173.060,35.859,156.728
C03549=1057.290,297.213,398.329,173.063,35.863,156.729
C03550=1057.296,297.461,398.296,173.067,35.867,156.730
C03551=1057.302,297.709,398.264,173.069,35.871,156.731
C03552=1057.308,297.957,398.231,173.073,35.875,156.732
C03553=1057.314,298.204,398.200,173.076,35.879,156.733
C03554=1057.320,298.452,398.168,173.080,35.883,156.734
C03555=1057.327,298.700,398.136,173.082,35.886,156.734
C03556=1057.333,298.948,398.104,173.085,35.891,156.735
C03557=1057.340,299.195,398.071,173.089,35.895,156.736
C03558=1057.346,299.444,398.039,173.092,35.899,156.737
C03559=1057.352,299.691,398.007,173.095,35.902,156.738
C03560=1057.358,299.939,397.975,173.098,35.906,156.739
C03561=1057.364,300.187,397.942,173.101,35.910,156.739
C03562=1057.371,300.434,397.910,173.105,35.914,156.740
C03563=1057.377,300.683,397.878,173.107,35.918,156.741
C03564=1057.383,300.930,397.845,173.111,35.922,156.742
C03565=1057.389,301.178,397.813,173.114,35.926,156.743
C03566=1057.396,301.426,397.780,173.118,35.930,156.744
C03567=1057.403,301.673,397.748,173.120,35.934,156.744
C03568=1057.409,301.921,397.716,173.123,35.938,156.745
C03569=1057.415,302.169,397.683,173.127,35.942,156.746
C03570=1057.421,302.417,397.651,173.130,35.946,156.747
C03571=1057.427,302.665,397.619,173.133,35.949,156.748
C03572=1057.434,302.912,397.586,173.136,35.953,156.749
C03573=1057.441,303.160,397.554,173.140,35.957,156.750
C03574=1057.447,303.407,397.521,173.143,35.962,156.750
C03575=1057.453,303.655,397.489,173.147,35.965,156.751
C03576=1057.460,303.909,397.455,173.150,35.969,156.752
C03577=1057.466,304.162,397.422,173.152,35.973,156.753
C03578=1057.473,304.415,397.389,173.156,35.977,156.754
C03579=1057.480,304.668,397.356,173.159,35.981,156.755
C03580=1057.486,304.916,397.323,173.163,35.985,156.756
C03581=1057.493,305.164,397.290,173.166,35.989,156.757
C03582=1057.499,305.411,397.258,173.170,35.994,156.757
C03583=1057.505,305.659,397.225,173.172,35.997,156.758
C03584=1057.512,305.906,397.192,173.176,36.001,156.759
C03585=1057.518,306.154,397.161,173.179,36.005,156.760
C03586=1057.525,306.403,397.127,173.182,36.009,156.761
C03587=1057.531,306.650,397.095,173.186,36.013,156.762
C03588=1057.538,306.898,397.062,173.189,36.017,156.763
C03589=1057.544,307.145,397.029,173.193,36.021,156.763
C03590=1057.550,307.393,396.997,173.195,36.025,156.764
C03591=1057.557,307.641,396.963,173.199,36.029,156.765
C03592=1057.563,307.889,396.931,173.202,36.033,156.766
C03593=1057.571,308.136,396.899,173.206,36.037,156.767
C03594=1057.577,308.384,396.866,173.209,36.041,156.768
C03595=1057.584,308.632,396.833,173.212,36.045,156.768
C03596=1057.590,308.879,396.799,173.216,36.049,156.769
C03597=1057.597,309.127,396.766,173.219,36.053,156.770
C03598=1057.603,309.375,396.733,173.223,36.057,156.771
C03599=1057.610,309.622,396.701,173.225,36.061,156.772
C03600=1057.616,309.870,396.668,173.229,36.065,156.773
C03601=1057.622,310.118,396.635,173.232,36.069,156.774
C03602=1057.629,310.366,396.602,173.236,36.073,156.775
C03603=1057.636,310.613,396.569,173.239,36.077,156.776
C03604=1057.644,310.861,396.536,173.243,36.080,156.776
C03605=1057.650,311.108,396.503,173.246,36.084,156.777
C03606=1057.656,311.356,396.471,173.250,36.089,156.778
C03607=1057.663,311.604,396.437,173.253,36.093,156.779
C03608=1057.670,311.851,396.404,173.256,36.097,156.780
C03609=1057.676,312.099,396.371,173.260,36.101,156.781
C03610=1057.683,312.347,396.338,173.263,36.105,156.782
C03611=1057.689,312.594,396.305,173.267,36.109,156.782
C03612=1057.696,312.842,396.272,173.270,36.113,156.783
C03613=1057.703,313.090,396.239,173.274,36.117,156.784
C03614=1057.709,313.338,396.206,173.276,36.121,156.785
C03615=1057.716,313.585,396.172,173.280,36.125,156.786
C03616=1057.722,313.833,396.139,173.283,36.129,156.787
C03617=1057.729,314.081,396.105,173.287,36.133,156.788
C03618=1057.735,314.328,396.072,173.290,36.137,156.789
C03619=1057.741,314.576,396.038,173.294,36.142,156.790
C03620=1057.748,314.824,396.005,173.297,36.146,156.791
C03621=1057.754,315.071,395.971,173.301,36.150,156.791
C03622=1057.761,315.319,395.937,173.304,36.154,156.792
C03623=1057.766,315.567,395.904,173.308,36.158,156.793
C03624=1057.773,315.814,395.871,173.311,36.162,156.794
C03625=1057.779,316.063,395.837,173.315,36.166,156.795
C03626=1057.786,316.309,395.803,173.318,36.170,156.796
C03627=1057.792,316.557,395.769,173.322,36.175,156.797
C03628=1057.799,316.805,395.736,173.325,36.179,156.798
C03629=1057.804,317.052,395.702,173.329,36.183,156.799
C03630=1057.812,317.300,395.668,173.332,36.188,156.800
C03631=1057.817,317.548,395.635,173.336,36.192,156.801
C03632=1057.824,317.805,395.600,173.339,36.196,156.802
C03633=1057.831,318.062,395.565,173.343,36.200,156.803
C03634=1057.838,318.319,395.529,173.346,36.205,156.804
C03635=1057.844,318.577,395.495,173.350,36.209,156.805
C03636=1057.851,318.825,395.460,173.353,36.214,156.806
C03637=1057.858,319.072,395.427,173.357,36.218,156.806
C03638=1057.864,319.320,395.393,173.360,36.222,156.807
C03639=1057.871,319.567,395.359,173.364,36.226,156.808
C03640=1057.877,319.815,395.325,173.368,36.230,156.809
